KUKA KRL program: EPS_2_25452_SANMH01_A_20260112013754.src

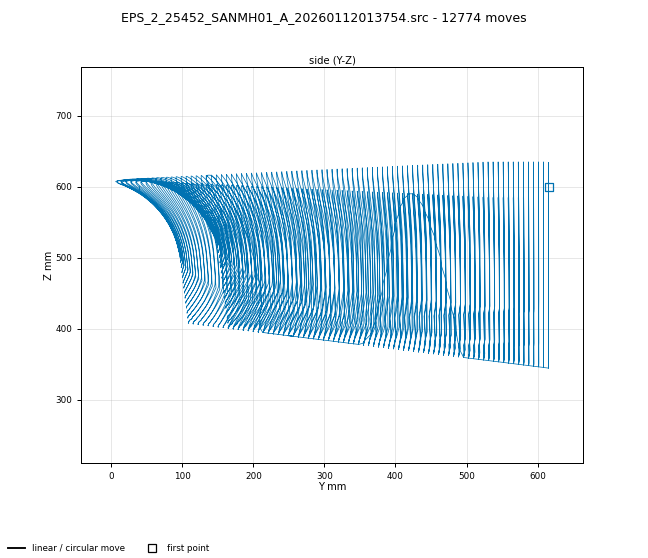
[picture p0: tool path of EPS_2_25452_SANMH01_A_20260112013754.src, 12774 of 12776 moves have a stored position in this frame; points joined in program order, loops and branches not executed]
&ACCESS RVP
&REL 4
&COMMENT QRS 19112012
&PARAM EDITMASK = *
DEF PART()
EXT BAS (BAS_COMMAND :IN,REAL :IN )
INT I
BAS (#INITMOV,0 )

;KUKA QRS Post kuka4.cps  Date:22-06-2017 !

File_ID=2960

QRS_PRE_INIT()

;Init var - Until changes are made in qrs_pre_init
Outlet_Square_prg=0
Inlet_1_Square_prg=0
Inlet_2_Square_prg=0
Inlet_3_Square_prg=0
Inlet_4_Square_prg=0
Inlet_5_Square_prg=0

Outlet_1={X 0.000, Y 530.070, Z 534.500, B 0.000, E1 0.000 }
Inlet_1={X 0.000, Y 533.640, Z 484.500, B 0.000, E1 171.000 }
Outlet_1_type=201
Inlet_1_type=201
;QRS#1=Sidecore dimensions
;QRS#2=200-8" PVC SDR 35
;QRS#3=200-8" PVC SDR 35
;QRS#4=
;QRS#5=
;QRS#6=
;QRS#7=
;QRS#8=
;QRS#9=12-08 PSX
;QRS#10=12-08 PSX
;QRS#11=
;QRS#12=
;QRS#13=
;QRS#14=
;QRS#15=
;QRS#16=1220x127x914 3'
;QRS#17=EPS Height
;QRS#18=635
;QRS#19=*
;QRS#20= UPDATED VERSION 22-06-2017
;QRS#21=*
Outlet_Square=0100
Inlet_1_Square=0100
Inlet_2_Square=0
Inlet_3_Square=0
Inlet_4_Square=0
Inlet_5_Square=0
Mill_Square=1
Outlet_Square_Prg=204
Inlet_1_Square_prg=204

QRS_INIT()

$ADVANCE=5

; T1
PTP {E1 173.589,E2 173.589}
PTP {X 0,Y 615.512,A -85,B 0,C 180,E1 173.589,E2 173.589,E3 0,E4 0,E5 0,E6 0}
QRS_SPEED_INIT()
LIN {X 0,Y 615.512,Z 600,A -85,B 0,C 180,E1 173.589,E2 173.589,E3 0,E4 0,E5 0,E6 0} C_VEL
LIN {X 0,Y 615.512,Z 354.868,A -85,B 0,C 180,E1 173.589,E2 173.589} C_VEL
LIN {X 0,Y 615.512,Z 346.696,A -85,B 0,C 180,E1 173.589,E2 173.589} C_VEL
LIN {X 0,Y 615.496,Z 344.696,A -85,B 0,C 180,E1 173.403,E2 173.403} C_VEL
LIN {X 0,Y 615.484,Z 344.688,A -85,B 0,C 180,E1 170.801,E2 170.801} C_VEL
LIN {X 0,Y 615.478,Z 344.686,A -85,B 0,C 180,E1 168.139,E2 168.139} C_VEL
LIN {X 0,Y 615.493,Z 344.701,A -85,B 0,C 180,E1 165.451,E2 165.451} C_VEL
LIN {X 0,Y 615.489,Z 344.683,A -85,B 0,C 180,E1 162.729,E2 162.729} C_VEL
LIN {X 0,Y 615.479,Z 344.691,A -85,B 0,C 180,E1 159.967,E2 159.967} C_VEL
LIN {X 0,Y 615.493,Z 344.699,A -85,B 0,C 180,E1 157.65,E2 157.65} C_VEL
LIN {X 0,Y 615.476,Z 344.688,A -85,B 0,C 180,E1 155.007,E2 155.007} C_VEL
LIN {X 0,Y 615.481,Z 344.684,A -85,B 0,C 180,E1 152.822,E2 152.822} C_VEL
LIN {X 0,Y 615.477,Z 344.691,A -85,B 0,C 180,E1 150.205,E2 150.205} C_VEL
LIN {X 0,Y 615.489,Z 344.694,A -85,B 0,C 180,E1 147.542,E2 147.542} C_VEL
LIN {X 0,Y 615.477,Z 344.687,A -85,B 0,C 180,E1 145.184,E2 145.184} C_VEL
LIN {X 0,Y 615.489,Z 344.683,A -85,B 0,C 180,E1 142.757,E2 142.757} C_VEL
LIN {X 0,Y 615.498,Z 344.699,A -85,B 0,C 180,E1 139.908,E2 139.908} C_VEL
LIN {X 0,Y 615.493,Z 344.69,A -85,B 0,C 180,E1 137.647,E2 137.647} C_VEL
LIN {X 0,Y 615.481,Z 344.684,A -85,B 0,C 180,E1 134.93,E2 134.93} C_VEL
LIN {X 0,Y 615.498,Z 344.7,A -85,B 0,C 180,E1 132.081,E2 132.081} C_VEL
LIN {X 0,Y 615.495,Z 344.688,A -85,B 0,C 180,E1 129.748,E2 129.748} C_VEL
LIN {X 0,Y 615.484,Z 344.685,A -85,B 0,C 180,E1 126.935,E2 126.935} C_VEL
LIN {X 0,Y 615.493,Z 344.693,A -85,B 0,C 180,E1 124.021,E2 124.021} C_VEL
LIN {X 0,Y 615.487,Z 344.685,A -85,B 0,C 180,E1 121.685,E2 121.685} C_VEL
LIN {X 0,Y 615.477,Z 344.685,A -85,B 0,C 180,E1 119.406,E2 119.406} C_VEL
LIN {X 0,Y 615.491,Z 344.805,A -85,B 0,C 180,E1 116.968,E2 116.968} C_VEL
LIN {X 0,Y 615.483,Z 360.204,A -85,B 0,C 180,E1 114.272,E2 114.272} C_VEL
LIN {X 0,Y 615.497,Z 374.44,A -85,B 0,C 180,E1 111.805,E2 111.805} C_VEL
LIN {X 0,Y 615.478,Z 480.331,A -85,B 0,C 180,E1 110.553,E2 110.553} C_VEL
LIN {X 0,Y 615.475,Z 493.827,A -85,B 0,C 180,E1 110.26,E2 110.26} C_VEL
LIN {X 0,Y 615.497,Z 506.182,A -85,B 0,C 180,E1 109.858,E2 109.858} C_VEL
LIN {X 0,Y 615.477,Z 518.044,A -85,B 0,C 180,E1 109.338,E2 109.338} C_VEL
LIN {X 0,Y 615.488,Z 528.758,A -85,B 0,C 180,E1 108.732,E2 108.732} C_VEL
LIN {X 0,Y 615.499,Z 539.692,A -85,B 0,C 180,E1 107.956,E2 107.956} C_VEL
LIN {X 0,Y 615.497,Z 549.463,A -85,B 0,C 180,E1 107.099,E2 107.099} C_VEL
LIN {X 0,Y 615.497,Z 557.985,A -85,B 0,C 180,E1 106.168,E2 106.168} C_VEL
LIN {X 0,Y 615.497,Z 565.024,A -85,B 0,C 180,E1 105.225,E2 105.225} C_VEL
LIN {X 0,Y 615.497,Z 570.956,A -85,B 0,C 180,E1 104.241,E2 104.241} C_VEL
LIN {X 0,Y 615.496,Z 575.897,A -85,B 0,C 180,E1 103.201,E2 103.201} C_VEL
LIN {X 0,Y 615.497,Z 579.504,A -85,B 0,C 180,E1 102.195,E2 102.195} C_VEL
LIN {X 0,Y 615.495,Z 582.657,A -85,B 0,C 180,E1 100.889,E2 100.889} C_VEL
LIN {X 0,Y 615.499,Z 583.995,A -85,B 0,C 180,E1 99.862,E2 99.862} C_VEL
LIN {X 0,Y 615.495,Z 584.296,A -85,B 0,C 180,E1 98.536,E2 98.536} C_VEL
LIN {X 0,Y 615.497,Z 583.85,A -85,B 0,C 180,E1 97.875,E2 97.875} C_VEL
LIN {X 0,Y 615.496,Z 581.72,A -85,B 0,C 180,E1 96.556,E2 96.556} C_VEL
LIN {X 0,Y 615.498,Z 579.037,A -85,B 0,C 180,E1 95.57,E2 95.57} C_VEL
LIN {X 0,Y 615.495,Z 575.36,A -85,B 0,C 180,E1 94.584,E2 94.584} C_VEL
LIN {X 0,Y 615.496,Z 570.584,A -85,B 0,C 180,E1 93.601,E2 93.601} C_VEL
LIN {X 0,Y 615.497,Z 564.573,A -85,B 0,C 180,E1 92.618,E2 92.618} C_VEL
LIN {X 0,Y 615.498,Z 557.116,A -85,B 0,C 180,E1 91.636,E2 91.636} C_VEL
LIN {X 0,Y 615.498,Z 549.527,A -85,B 0,C 180,E1 90.818,E2 90.818} C_VEL
LIN {X 0,Y 615.498,Z 539.238,A -85,B 0,C 180,E1 89.918,E2 89.918} C_VEL
LIN {X 0,Y 615.484,Z 528.822,A -85,B 0,C 180,E1 89.182,E2 89.182} C_VEL
LIN {X 0,Y 615.482,Z 517.116,A -85,B 0,C 180,E1 88.528,E2 88.528} C_VEL
LIN {X 0,Y 615.495,Z 504.679,A -85,B 0,C 180,E1 87.996,E2 87.996} C_VEL
LIN {X 0,Y 615.476,Z 493.022,A -85,B 0,C 180,E1 87.628,E2 87.628} C_VEL
LIN {X 0,Y 615.478,Z 480.616,A -85,B 0,C 180,E1 87.362,E2 87.362} C_VEL
LIN {X 0,Y 615.491,Z 374.366,A -85,B 0,C 180,E1 86.092,E2 86.092} C_VEL
LIN {X 0,Y 615.486,Z 358.994,A -85,B 0,C 180,E1 83.428,E2 83.428} C_VEL
LIN {X 0,Y 615.486,Z 344.686,A -85,B 0,C 180,E1 80.905,E2 80.905} C_VEL
LIN {X 0,Y 615.487,Z 344.686,A -85,B 0,C 180,E1 78.139,E2 78.139} C_VEL
LIN {X 0,Y 615.495,Z 344.696,A -85,B 0,C 180,E1 75.451,E2 75.451} C_VEL
LIN {X 0,Y 615.478,Z 344.685,A -85,B 0,C 180,E1 72.73,E2 72.73} C_VEL
LIN {X 0,Y 615.494,Z 344.692,A -85,B 0,C 180,E1 69.968,E2 69.968} C_VEL
LIN {X 0,Y 615.489,Z 344.685,A -85,B 0,C 180,E1 67.156,E2 67.156} C_VEL
LIN {X 0,Y 615.489,Z 344.688,A -85,B 0,C 180,E1 64.285,E2 64.285} C_VEL
LIN {X 0,Y 615.49,Z 344.687,A -85,B 0,C 180,E1 61.343,E2 61.343} C_VEL
LIN {X 0,Y 615.482,Z 344.684,A -85,B 0,C 180,E1 58.916,E2 58.916} C_VEL
LIN {X 0,Y 615.497,Z 344.7,A -85,B 0,C 180,E1 55.98,E2 55.98} C_VEL
LIN {X 0,Y 615.483,Z 344.684,A -85,B 0,C 180,E1 53.065,E2 53.065} C_VEL
LIN {X 0,Y 615.494,Z 344.695,A -85,B 0,C 180,E1 50.251,E2 50.251} C_VEL
LIN {X 0,Y 615.476,Z 344.691,A -85,B 0,C 180,E1 47.647,E2 47.647} C_VEL
LIN {X 0,Y 615.479,Z 344.685,A -85,B 0,C 180,E1 44.932,E2 44.932} C_VEL
LIN {X 0,Y 615.486,Z 344.698,A -85,B 0,C 180,E1 42.082,E2 42.082} C_VEL
LIN {X 0,Y 615.477,Z 344.69,A -85,B 0,C 180,E1 39.751,E2 39.751} C_VEL
LIN {X 0,Y 615.478,Z 344.687,A -85,B 0,C 180,E1 36.937,E2 36.937} C_VEL
LIN {X 0,Y 615.481,Z 344.693,A -85,B 0,C 180,E1 34.023,E2 34.023} C_VEL
LIN {X 0,Y 615.479,Z 344.686,A -85,B 0,C 180,E1 31.686,E2 31.686} C_VEL
LIN {X 0,Y 615.486,Z 344.683,A -85,B 0,C 180,E1 29.407,E2 29.407} C_VEL
LIN {X 0,Y 615.495,Z 344.699,A -85,B 0,C 180,E1 26.444,E2 26.444} C_VEL
LIN {X 0,Y 615.486,Z 344.683,A -85,B 0,C 180,E1 23.557,E2 23.557} C_VEL
LIN {X 0,Y 615.486,Z 344.698,A -85,B 0,C 180,E1 20.731,E2 20.731} C_VEL
LIN {X 0,Y 615.477,Z 344.687,A -85,B 0,C 180,E1 17.958,E2 17.958} C_VEL
LIN {X 0,Y 615.491,Z 344.686,A -85,B 0,C 180,E1 15.226,E2 15.226} C_VEL
LIN {X 0,Y 615.493,Z 344.694,A -85,B 0,C 180,E1 12.53,E2 12.53} C_VEL
LIN {X 0,Y 615.477,Z 344.685,A -85,B 0,C 180,E1 9.863,E2 9.863} C_VEL
LIN {X 0,Y 615.49,Z 344.69,A -85,B 0,C 180,E1 7.216,E2 7.216} C_VEL
LIN {X 0,Y 615.493,Z 344.691,A -85,B 0,C 180,E1 4.585,E2 4.585} C_VEL
LIN {X 0,Y 615.477,Z 344.685,A -85,B 0,C 180,E1 1.963,E2 1.963} C_VEL
LIN {X 0,Y 615.493,Z 344.69,A -85,B 0,C 180,E1 -0.654,E2 -0.654} C_VEL
LIN {X 0,Y 615.491,Z 344.691,A -85,B 0,C 180,E1 -3.273,E2 -3.273} C_VEL
LIN {X 0,Y 615.476,Z 344.685,A -85,B 0,C 180,E1 -5.899,E2 -5.899} C_VEL
LIN {X 0,Y 615.493,Z 344.691,A -85,B 0,C 180,E1 -8.536,E2 -8.536} C_VEL
LIN {X 0,Y 615.49,Z 344.69,A -85,B 0,C 180,E1 -11.193,E2 -11.193} C_VEL
LIN {X 0,Y 615.474,Z 344.686,A -85,B 0,C 180,E1 -13.933,E2 -13.933} C_VEL
LIN {X 0,Y 615.496,Z 344.696,A -85,B 0,C 180,E1 -16.586,E2 -16.586} C_VEL
LIN {X 0,Y 615.488,Z 344.685,A -85,B 0,C 180,E1 -19.338,E2 -19.338} C_VEL
LIN {X 0,Y 615.48,Z 344.69,A -85,B 0,C 180,E1 -22.137,E2 -22.137} C_VEL
LIN {X 0,Y 615.484,Z 344.69,A -85,B 0,C 180,E1 -24.992,E2 -24.992} C_VEL
LIN {X 0,Y 615.483,Z 344.686,A -85,B 0,C 180,E1 -27.177,E2 -27.177} C_VEL
LIN {X 0,Y 615.477,Z 344.687,A -85,B 0,C 180,E1 -29.795,E2 -29.795} C_VEL
LIN {X 0,Y 615.496,Z 344.7,A -85,B 0,C 180,E1 -32.457,E2 -32.457} C_VEL
LIN {X 0,Y 615.48,Z 344.691,A -85,B 0,C 180,E1 -34.816,E2 -34.816} C_VEL
LIN {X 0,Y 615.489,Z 344.682,A -85,B 0,C 180,E1 -37.242,E2 -37.242} C_VEL
LIN {X 0,Y 615.486,Z 344.696,A -85,B 0,C 180,E1 -40.09,E2 -40.09} C_VEL
LIN {X 0,Y 615.493,Z 344.697,A -85,B 0,C 180,E1 -42.353,E2 -42.353} C_VEL
LIN {X 0,Y 615.48,Z 344.684,A -85,B 0,C 180,E1 -45.069,E2 -45.069} C_VEL
LIN {X 0,Y 615.486,Z 344.696,A -85,B 0,C 180,E1 -47.92,E2 -47.92} C_VEL
LIN {X 0,Y 615.494,Z 344.695,A -85,B 0,C 180,E1 -50.252,E2 -50.252} C_VEL
LIN {X 0,Y 615.483,Z 344.684,A -85,B 0,C 180,E1 -53.064,E2 -53.064} C_VEL
LIN {X 0,Y 615.494,Z 344.701,A -85,B 0,C 180,E1 -55.979,E2 -55.979} C_VEL
LIN {X 0,Y 615.482,Z 344.684,A -85,B 0,C 180,E1 -58.915,E2 -58.915} C_VEL
LIN {X 0,Y 615.485,Z 344.692,A -85,B 0,C 180,E1 -61.551,E2 -61.551} C_VEL
LIN {X 0,Y 615.481,Z 344.687,A -85,B 0,C 180,E1 -64.433,E2 -64.433} C_VEL
LIN {X 0,Y 615.487,Z 344.827,A -85,B 0,C 180,E1 -67.067,E2 -67.067} C_VEL
LIN {X 0,Y 615.484,Z 366.758,A -85,B 0,C 180,E1 -69.968,E2 -69.968} C_VEL
LIN {X 0,Y 615.478,Z 388,A -85,B 0,C 180,E1 -72.73,E2 -72.73} C_VEL
LIN {X 0,Y 615.479,Z 409.218,A -85,B 0,C 180,E1 -75.451,E2 -75.451} C_VEL
LIN {X 0,Y 615.497,Z 422.298,A -85,B 0,C 180,E1 -77.114,E2 -77.114} C_VEL
LIN {X 0,Y 615.479,Z 530.847,A -85,B 0,C 180,E1 -78.411,E2 -78.411} C_VEL
LIN {X 0,Y 615.478,Z 543.355,A -85,B 0,C 180,E1 -78.682,E2 -78.682} C_VEL
LIN {X 0,Y 615.491,Z 556.568,A -85,B 0,C 180,E1 -79.111,E2 -79.111} C_VEL
LIN {X 0,Y 615.478,Z 568.483,A -85,B 0,C 180,E1 -79.639,E2 -79.639} C_VEL
LIN {X 0,Y 615.487,Z 579.999,A -85,B 0,C 180,E1 -80.304,E2 -80.304} C_VEL
LIN {X 0,Y 615.499,Z 590.344,A -85,B 0,C 180,E1 -81.05,E2 -81.05} C_VEL
LIN {X 0,Y 615.497,Z 598.814,A -85,B 0,C 180,E1 -81.794,E2 -81.794} C_VEL
LIN {X 0,Y 615.498,Z 606.608,A -85,B 0,C 180,E1 -82.62,E2 -82.62} C_VEL
LIN {X 0,Y 615.496,Z 614.204,A -85,B 0,C 180,E1 -83.608,E2 -83.608} C_VEL
LIN {X 0,Y 615.498,Z 621.205,A -85,B 0,C 180,E1 -84.759,E2 -84.759} C_VEL
LIN {X 0,Y 615.493,Z 625.852,A -85,B 0,C 180,E1 -85.744,E2 -85.744} C_VEL
LIN {X 0,Y 615.495,Z 629.399,A -85,B 0,C 180,E1 -86.727,E2 -86.727} C_VEL
LIN {X 0,Y 615.497,Z 631.233,A -85,B 0,C 180,E1 -87.382,E2 -87.382} C_VEL
LIN {X 0,Y 615.497,Z 632.608,A -85,B 0,C 180,E1 -88.037,E2 -88.037} C_VEL
LIN {X 0,Y 615.496,Z 634.174,A -85,B 0,C 180,E1 -89.346,E2 -89.346} C_VEL
LIN {X 0,Y 615.494,Z 634.389,A -85,B 0,C 180,E1 -90,E2 -90} C_VEL
LIN {X 0,Y 615.496,Z 633.58,A -85,B 0,C 180,E1 -91.309,E2 -91.309} C_VEL
LIN {X 0,Y 615.497,Z 632.608,A -85,B 0,C 180,E1 -91.963,E2 -91.963} C_VEL
LIN {X 0,Y 615.497,Z 631.233,A -85,B 0,C 180,E1 -92.618,E2 -92.618} C_VEL
LIN {X 0,Y 615.496,Z 628.35,A -85,B 0,C 180,E1 -93.601,E2 -93.601} C_VEL
LIN {X 0,Y 615.498,Z 624.442,A -85,B 0,C 180,E1 -94.584,E2 -94.584} C_VEL
LIN {X 0,Y 615.499,Z 619.406,A -85,B 0,C 180,E1 -95.57,E2 -95.57} C_VEL
LIN {X 0,Y 615.497,Z 612.869,A -85,B 0,C 180,E1 -96.583,E2 -96.583} C_VEL
LIN {X 0,Y 615.497,Z 605.135,A -85,B 0,C 180,E1 -97.545,E2 -97.545} C_VEL
LIN {X 0,Y 615.498,Z 597.047,A -85,B 0,C 180,E1 -98.371,E2 -98.371} C_VEL
LIN {X 0,Y 615.499,Z 587.17,A -85,B 0,C 180,E1 -99.198,E2 -99.198} C_VEL
LIN {X 0,Y 615.488,Z 575.985,A -85,B 0,C 180,E1 -99.945,E2 -99.945} C_VEL
LIN {X 0,Y 615.481,Z 565.029,A -85,B 0,C 180,E1 -100.527,E2 -100.527} C_VEL
LIN {X 0,Y 615.49,Z 552.452,A -85,B 0,C 180,E1 -101.041,E2 -101.041} C_VEL
LIN {X 0,Y 615.477,Z 540.079,A -85,B 0,C 180,E1 -101.401,E2 -101.401} C_VEL
LIN {X 0,Y 615.481,Z 526.487,A -85,B 0,C 180,E1 -101.652,E2 -101.652} C_VEL
LIN {X 0,Y 615.497,Z 422.298,A -85,B 0,C 180,E1 -102.886,E2 -102.886} C_VEL
LIN {X 0,Y 615.485,Z 399.937,A -85,B 0,C 180,E1 -105.735,E2 -105.735} C_VEL
LIN {X 0,Y 615.481,Z 377.716,A -85,B 0,C 180,E1 -108.602,E2 -108.602} C_VEL
LIN {X 0,Y 615.478,Z 357.457,A -85,B 0,C 180,E1 -111.256,E2 -111.256} C_VEL
LIN {X 0,Y 615.486,Z 344.684,A -85,B 0,C 180,E1 -112.977,E2 -112.977} C_VEL
LIN {X 0,Y 615.489,Z 344.689,A -85,B 0,C 180,E1 -115.715,E2 -115.715} C_VEL
LIN {X 0,Y 615.488,Z 344.686,A -85,B 0,C 180,E1 -118.657,E2 -118.657} C_VEL
LIN {X 0,Y 615.482,Z 344.684,A -85,B 0,C 180,E1 -121.085,E2 -121.085} C_VEL
LIN {X 0,Y 615.494,Z 344.7,A -85,B 0,C 180,E1 -124.021,E2 -124.021} C_VEL
LIN {X 0,Y 615.483,Z 344.684,A -85,B 0,C 180,E1 -126.936,E2 -126.936} C_VEL
LIN {X 0,Y 615.494,Z 344.697,A -85,B 0,C 180,E1 -129.748,E2 -129.748} C_VEL
LIN {X 0,Y 615.478,Z 344.689,A -85,B 0,C 180,E1 -132.353,E2 -132.353} C_VEL
LIN {X 0,Y 615.48,Z 344.686,A -85,B 0,C 180,E1 -135.068,E2 -135.068} C_VEL
LIN {X 0,Y 615.486,Z 344.696,A -85,B 0,C 180,E1 -137.918,E2 -137.918} C_VEL
LIN {X 0,Y 615.477,Z 344.689,A -85,B 0,C 180,E1 -140.249,E2 -140.249} C_VEL
LIN {X 0,Y 615.482,Z 344.688,A -85,B 0,C 180,E1 -143.062,E2 -143.062} C_VEL
LIN {X 0,Y 615.481,Z 344.691,A -85,B 0,C 180,E1 -145.978,E2 -145.978} C_VEL
LIN {X 0,Y 615.479,Z 344.685,A -85,B 0,C 180,E1 -148.314,E2 -148.314} C_VEL
LIN {X 0,Y 615.487,Z 344.683,A -85,B 0,C 180,E1 -150.594,E2 -150.594} C_VEL
LIN {X 0,Y 615.497,Z 344.695,A -85,B 0,C 180,E1 -153.556,E2 -153.556} C_VEL
LIN {X 0,Y 615.486,Z 344.683,A -85,B 0,C 180,E1 -156.444,E2 -156.444} C_VEL
LIN {X 0,Y 615.495,Z 344.701,A -85,B 0,C 180,E1 -159.27,E2 -159.27} C_VEL
LIN {X 0,Y 615.477,Z 344.686,A -85,B 0,C 180,E1 -162.043,E2 -162.043} C_VEL
LIN {X 0,Y 615.492,Z 344.689,A -85,B 0,C 180,E1 -164.774,E2 -164.774} C_VEL
LIN {X 0,Y 615.491,Z 344.69,A -85,B 0,C 180,E1 -167.47,E2 -167.47} C_VEL
LIN {X 0,Y 615.477,Z 344.685,A -85,B 0,C 180,E1 -170.138,E2 -170.138} C_VEL
LIN {X 0,Y 615.495,Z 344.693,A -85,B 0,C 180,E1 -172.785,E2 -172.785} C_VEL
LIN {X 0,Y 615.491,Z 344.688,A -85,B 0,C 180,E1 -175.416,E2 -175.416} C_VEL
LIN {X 0,Y 615.477,Z 344.685,A -85,B 0,C 180,E1 -178.037,E2 -178.037} C_VEL
LIN {X 0,Y 615.495,Z 344.694,A -85,B 0,C 180,E1 -180.654,E2 -180.654} C_VEL
LIN {X 0,Y 615.491,Z 344.687,A -85,B 0,C 180,E1 -183.273,E2 -183.273} C_VEL
LIN {X 0,Y 615.476,Z 344.686,A -85,B 0,C 180,E1 -185.899,E2 -185.899} C_VEL
LIN {X 0,Y 615.496,Z 344.696,A -85,B 0,C 180,E1 -186.597,E2 -186.597} C_VEL
LIN {X 0,Y 614.815,Z 344.835,A -85,B 0,C 180,E1 -187.143,E2 -187.143} C_VEL
LIN {X 0,Y 611.975,Z 345.25,A -85,B 0,C 180,E1 -188.028,E2 -188.028} C_VEL
LIN {X 0,Y 609.58,Z 345.56,A -85,B 0,C 180,E1 -188.741,E2 -188.741} C_VEL
LIN {X 0,Y 608.544,Z 345.678,A -85,B 0,C 180,E1 -189.291,E2 -189.291} C_VEL
LIN {X 0,Y 608.454,Z 345.688,A -85,B 0,C 180,E1 -189.477,E2 -189.477} C_VEL
LIN {X 0,Y 608.456,Z 345.689,A -85,B 0,C 180,E1 -192,E2 -192} C_VEL
LIN {X 0,Y 608.478,Z 345.692,A -85,B 0,C 180,E1 -194.721,E2 -194.721} C_VEL
LIN {X 0,Y 608.451,Z 345.688,A -85,B 0,C 180,E1 -197.477,E2 -197.477} C_VEL
LIN {X 0,Y 608.46,Z 345.694,A -85,B 0,C 180,E1 -200.275,E2 -200.275} C_VEL
LIN {X 0,Y 608.456,Z 345.697,A -85,B 0,C 180,E1 -202.479,E2 -202.479} C_VEL
LIN {X 0,Y 608.45,Z 345.695,A -85,B 0,C 180,E1 -204.572,E2 -204.572} C_VEL
LIN {X 0,Y 608.473,Z 345.685,A -85,B 0,C 180,E1 -207.209,E2 -207.209} C_VEL
LIN {X 0,Y 608.461,Z 345.692,A -85,B 0,C 180,E1 -209.973,E2 -209.973} C_VEL
LIN {X 0,Y 608.462,Z 345.691,A -85,B 0,C 180,E1 -212.525,E2 -212.525} C_VEL
LIN {X 0,Y 608.439,Z 345.689,A -85,B 0,C 180,E1 -215.278,E2 -215.278} C_VEL
LIN {X 0,Y 608.473,Z 345.69,A -85,B 0,C 180,E1 -217.747,E2 -217.747} C_VEL
LIN {X 0,Y 608.478,Z 345.69,A -85,B 0,C 180,E1 -220.334,E2 -220.334} C_VEL
LIN {X 0,Y 608.484,Z 345.685,A -85,B 0,C 180,E1 -223.312,E2 -223.312} C_VEL
LIN {X 0,Y 608.477,Z 345.692,A -85,B 0,C 180,E1 -226.133,E2 -226.133} C_VEL
LIN {X 0,Y 608.45,Z 345.688,A -85,B 0,C 180,E1 -228.824,E2 -228.824} C_VEL
LIN {X 0,Y 608.473,Z 345.689,A -85,B 0,C 180,E1 -231.413,E2 -231.413} C_VEL
LIN {X 0,Y 608.48,Z 345.692,A -85,B 0,C 180,E1 -233.951,E2 -233.951} C_VEL
LIN {X 0,Y 608.463,Z 345.688,A -85,B 0,C 180,E1 -236.33,E2 -236.33} C_VEL
LIN {X 0,Y 608.448,Z 345.688,A -85,B 0,C 180,E1 -238.733,E2 -238.733} C_VEL
LIN {X 0,Y 608.482,Z 345.69,A -85,B 0,C 180,E1 -241.38,E2 -241.38} C_VEL
LIN {X 0,Y 608.479,Z 345.704,A -85,B 0,C 180,E1 -242.962,E2 -242.962} C_VEL
LIN {X 0,Y 608.478,Z 362.057,A -85,B 0,C 180,E1 -245.849,E2 -245.849} C_VEL
LIN {X 0,Y 608.467,Z 374.632,A -85,B 0,C 180,E1 -248.042,E2 -248.042} C_VEL
LIN {X 0,Y 608.53,Z 481.606,A -85,B 0,C 180,E1 -249.333,E2 -249.333} C_VEL
LIN {X 0,Y 608.52,Z 495.277,A -85,B 0,C 180,E1 -249.646,E2 -249.646} C_VEL
LIN {X 0,Y 608.52,Z 508.023,A -85,B 0,C 180,E1 -250.081,E2 -250.081} C_VEL
LIN {X 0,Y 608.505,Z 519.44,A -85,B 0,C 180,E1 -250.607,E2 -250.607} C_VEL
LIN {X 0,Y 608.471,Z 530.955,A -85,B 0,C 180,E1 -251.286,E2 -251.286} C_VEL
LIN {X 0,Y 608.478,Z 541.839,A -85,B 0,C 180,E1 -252.09,E2 -252.09} C_VEL
LIN {X 0,Y 608.462,Z 552.081,A -85,B 0,C 180,E1 -253.044,E2 -253.044} C_VEL
LIN {X 0,Y 608.462,Z 560.996,A -85,B 0,C 180,E1 -254.079,E2 -254.079} C_VEL
LIN {X 0,Y 608.451,Z 568.049,A -85,B 0,C 180,E1 -255.108,E2 -255.108} C_VEL
LIN {X 0,Y 608.432,Z 574.549,A -85,B 0,C 180,E1 -256.319,E2 -256.319} C_VEL
LIN {X 0,Y 608.428,Z 578.613,A -85,B 0,C 180,E1 -257.322,E2 -257.322} C_VEL
LIN {X 0,Y 608.445,Z 580.752,A -85,B 0,C 180,E1 -258,E2 -258} C_VEL
LIN {X 0,Y 608.423,Z 583.219,A -85,B 0,C 180,E1 -259.07,E2 -259.07} C_VEL
LIN {X 0,Y 608.434,Z 584.527,A -85,B 0,C 180,E1 -260.023,E2 -260.023} C_VEL
LIN {X 0,Y 608.419,Z 584.931,A -85,B 0,C 180,E1 -261.364,E2 -261.364} C_VEL
LIN {X 0,Y 608.422,Z 584.554,A -85,B 0,C 180,E1 -262.033,E2 -262.033} C_VEL
LIN {X 0,Y 608.421,Z 583.75,A -85,B 0,C 180,E1 -262.7,E2 -262.7} C_VEL
LIN {X 0,Y 608.449,Z 582.463,A -85,B 0,C 180,E1 -263.398,E2 -263.398} C_VEL
LIN {X 0,Y 608.442,Z 578.86,A -85,B 0,C 180,E1 -264.698,E2 -264.698} C_VEL
LIN {X 0,Y 608.441,Z 574.9,A -85,B 0,C 180,E1 -265.694,E2 -265.694} C_VEL
LIN {X 0,Y 608.458,Z 568.82,A -85,B 0,C 180,E1 -266.855,E2 -266.855} C_VEL
LIN {X 0,Y 608.454,Z 562.203,A -85,B 0,C 180,E1 -267.849,E2 -267.849} C_VEL
LIN {X 0,Y 608.479,Z 554.016,A -85,B 0,C 180,E1 -268.842,E2 -268.842} C_VEL
LIN {X 0,Y 608.469,Z 545.669,A -85,B 0,C 180,E1 -269.669,E2 -269.669} C_VEL
LIN {X 0,Y 608.479,Z 535.396,A -85,B 0,C 180,E1 -270.496,E2 -270.496} C_VEL
LIN {X 0,Y 608.485,Z 523.897,A -85,B 0,C 180,E1 -271.241,E2 -271.241} C_VEL
LIN {X 0,Y 608.502,Z 512.472,A -85,B 0,C 180,E1 -271.82,E2 -271.82} C_VEL
LIN {X 0,Y 608.512,Z 499.459,A -85,B 0,C 180,E1 -272.317,E2 -272.317} C_VEL
LIN {X 0,Y 608.521,Z 486.295,A -85,B 0,C 180,E1 -272.668,E2 -272.668} C_VEL
LIN {X 0,Y 608.536,Z 471.453,A -85,B 0,C 180,E1 -272.896,E2 -272.896} C_VEL
LIN {X 0,Y 608.537,Z 375.202,A -85,B 0,C 180,E1 -274.036,E2 -274.036} C_VEL
LIN {X 0,Y 608.458,Z 374.585,A -85,B 0,C 180,E1 -274.057,E2 -274.057} C_VEL
LIN {X 0,Y 608.486,Z 357.93,A -85,B 0,C 180,E1 -276.966,E2 -276.966} C_VEL
LIN {X 0,Y 608.477,Z 345.686,A -85,B 0,C 180,E1 -279.138,E2 -279.138} C_VEL
LIN {X 0,Y 608.465,Z 345.689,A -85,B 0,C 180,E1 -281.999,E2 -281.999} C_VEL
LIN {X 0,Y 608.48,Z 345.689,A -85,B 0,C 180,E1 -284.72,E2 -284.72} C_VEL
LIN {X 0,Y 608.452,Z 345.688,A -85,B 0,C 180,E1 -287.476,E2 -287.476} C_VEL
LIN {X 0,Y 608.47,Z 345.696,A -85,B 0,C 180,E1 -290.273,E2 -290.273} C_VEL
LIN {X 0,Y 608.451,Z 345.688,A -85,B 0,C 180,E1 -293.123,E2 -293.123} C_VEL
LIN {X 0,Y 608.472,Z 345.688,A -85,B 0,C 180,E1 -295.72,E2 -295.72} C_VEL
LIN {X 0,Y 608.476,Z 345.687,A -85,B 0,C 180,E1 -298.619,E2 -298.619} C_VEL
LIN {X 0,Y 608.447,Z 345.689,A -85,B 0,C 180,E1 -301.317,E2 -301.317} C_VEL
LIN {X 0,Y 608.473,Z 345.69,A -85,B 0,C 180,E1 -303.734,E2 -303.734} C_VEL
LIN {X 0,Y 608.479,Z 345.694,A -85,B 0,C 180,E1 -306.089,E2 -306.089} C_VEL
LIN {X 0,Y 608.471,Z 345.687,A -85,B 0,C 180,E1 -308.587,E2 -308.587} C_VEL
LIN {X 0,Y 608.457,Z 345.689,A -85,B 0,C 180,E1 -311.341,E2 -311.341} C_VEL
LIN {X 0,Y 608.449,Z 345.692,A -85,B 0,C 180,E1 -314.263,E2 -314.263} C_VEL
LIN {X 0,Y 608.453,Z 345.688,A -85,B 0,C 180,E1 -317.04,E2 -317.04} C_VEL
LIN {X 0,Y 608.449,Z 345.698,A -85,B 0,C 180,E1 -319.696,E2 -319.696} C_VEL
LIN {X 0,Y 608.467,Z 345.688,A -85,B 0,C 180,E1 -322.253,E2 -322.253} C_VEL
LIN {X 0,Y 608.436,Z 345.69,A -85,B 0,C 180,E1 -324.721,E2 -324.721} C_VEL
LIN {X 0,Y 608.466,Z 345.694,A -85,B 0,C 180,E1 -327.475,E2 -327.475} C_VEL
LIN {X 0,Y 608.462,Z 345.688,A -85,B 0,C 180,E1 -330.22,E2 -330.22} C_VEL
LIN {X 0,Y 608.475,Z 345.685,A -85,B 0,C 180,E1 -332.791,E2 -332.791} C_VEL
LIN {X 0,Y 608.453,Z 345.698,A -85,B 0,C 180,E1 -335.429,E2 -335.429} C_VEL
LIN {X 0,Y 608.47,Z 345.685,A -85,B 0,C 180,E1 -338.308,E2 -338.308} C_VEL
LIN {X 0,Y 608.472,Z 345.695,A -85,B 0,C 180,E1 -341.28,E2 -341.28} C_VEL
LIN {X 0,Y 608.457,Z 345.689,A -85,B 0,C 180,E1 -343.906,E2 -343.906} C_VEL
LIN {X 0,Y 608.464,Z 345.688,A -85,B 0,C 180,E1 -346.643,E2 -346.643} C_VEL
LIN {X 0,Y 608.474,Z 345.693,A -85,B 0,C 180,E1 -349.35,E2 -349.35} C_VEL
LIN {X 0,Y 608.471,Z 345.685,A -85,B 0,C 180,E1 -352.033,E2 -352.033} C_VEL
LIN {X 0,Y 608.469,Z 345.689,A -85,B 0,C 180,E1 -354.698,E2 -354.698} C_VEL
LIN {X 0,Y 608.485,Z 345.689,A -85,B 0,C 180,E1 -357.352,E2 -357.352} C_VEL
LIN {X 0,Y 608.468,Z 345.686,A -85,B 0,C 180,E1 -360,E2 -360} C_VEL
LIN {X 0,Y 608.485,Z 345.689,A -85,B 0,C 180,E1 -362.648,E2 -362.648} C_VEL
LIN {X 0,Y 608.47,Z 345.689,A -85,B 0,C 180,E1 -365.302,E2 -365.302} C_VEL
LIN {X 0,Y 608.471,Z 345.685,A -85,B 0,C 180,E1 -367.967,E2 -367.967} C_VEL
LIN {X 0,Y 608.473,Z 345.693,A -85,B 0,C 180,E1 -370.65,E2 -370.65} C_VEL
LIN {X 0,Y 608.464,Z 345.688,A -85,B 0,C 180,E1 -373.356,E2 -373.356} C_VEL
LIN {X 0,Y 608.457,Z 345.688,A -85,B 0,C 180,E1 -376.094,E2 -376.094} C_VEL
LIN {X 0,Y 608.456,Z 345.694,A -85,B 0,C 180,E1 -378.87,E2 -378.87} C_VEL
LIN {X 0,Y 608.47,Z 345.685,A -85,B 0,C 180,E1 -381.691,E2 -381.691} C_VEL
LIN {X 0,Y 608.453,Z 345.698,A -85,B 0,C 180,E1 -384.571,E2 -384.571} C_VEL
LIN {X 0,Y 608.475,Z 345.686,A -85,B 0,C 180,E1 -387.209,E2 -387.209} C_VEL
LIN {X 0,Y 608.46,Z 345.689,A -85,B 0,C 180,E1 -389.973,E2 -389.973} C_VEL
LIN {X 0,Y 608.468,Z 345.694,A -85,B 0,C 180,E1 -392.525,E2 -392.525} C_VEL
LIN {X 0,Y 608.438,Z 345.689,A -85,B 0,C 180,E1 -395.278,E2 -395.278} C_VEL
LIN {X 0,Y 608.467,Z 345.688,A -85,B 0,C 180,E1 -397.746,E2 -397.746} C_VEL
LIN {X 0,Y 608.449,Z 345.698,A -85,B 0,C 180,E1 -400.33,E2 -400.33} C_VEL
LIN {X 0,Y 608.483,Z 345.684,A -85,B 0,C 180,E1 -403.312,E2 -403.312} C_VEL
LIN {X 0,Y 608.467,Z 345.696,A -85,B 0,C 180,E1 -406.132,E2 -406.132} C_VEL
LIN {X 0,Y 608.45,Z 345.689,A -85,B 0,C 180,E1 -408.824,E2 -408.824} C_VEL
LIN {X 0,Y 608.47,Z 345.687,A -85,B 0,C 180,E1 -411.413,E2 -411.413} C_VEL
LIN {X 0,Y 608.478,Z 345.694,A -85,B 0,C 180,E1 -413.951,E2 -413.951} C_VEL
LIN {X 0,Y 608.463,Z 345.691,A -85,B 0,C 180,E1 -416.33,E2 -416.33} C_VEL
LIN {X 0,Y 608.476,Z 345.685,A -85,B 0,C 180,E1 -418.728,E2 -418.728} C_VEL
LIN {X 0,Y 608.474,Z 345.687,A -85,B 0,C 180,E1 -421.38,E2 -421.38} C_VEL
LIN {X 0,Y 608.471,Z 345.689,A -85,B 0,C 180,E1 -424.28,E2 -424.28} C_VEL
LIN {X 0,Y 608.479,Z 345.824,A -85,B 0,C 180,E1 -426.923,E2 -426.923} C_VEL
LIN {X 0,Y 608.582,Z 361.447,A -85,B 0,C 180,E1 -429.024,E2 -429.024} C_VEL
LIN {X 0,Y 608.518,Z 382.72,A -85,B 0,C 180,E1 -431.831,E2 -431.831} C_VEL
LIN {X 0,Y 608.492,Z 402.663,A -85,B 0,C 180,E1 -434.423,E2 -434.423} C_VEL
LIN {X 0,Y 608.503,Z 422.524,A -85,B 0,C 180,E1 -436.974,E2 -436.974} C_VEL
LIN {X 0,Y 608.538,Z 530.962,A -85,B 0,C 180,E1 -438.277,E2 -438.277} C_VEL
LIN {X 0,Y 608.514,Z 544.226,A -85,B 0,C 180,E1 -438.572,E2 -438.572} C_VEL
LIN {X 0,Y 608.517,Z 556.598,A -85,B 0,C 180,E1 -438.981,E2 -438.981} C_VEL
LIN {X 0,Y 608.498,Z 568.639,A -85,B 0,C 180,E1 -439.519,E2 -439.519} C_VEL
LIN {X 0,Y 608.48,Z 580.201,A -85,B 0,C 180,E1 -440.191,E2 -440.191} C_VEL
LIN {X 0,Y 608.485,Z 590.596,A -85,B 0,C 180,E1 -440.946,E2 -440.946} C_VEL
LIN {X 0,Y 608.475,Z 599.114,A -85,B 0,C 180,E1 -441.699,E2 -441.699} C_VEL
LIN {X 0,Y 608.471,Z 606.962,A -85,B 0,C 180,E1 -442.534,E2 -442.534} C_VEL
LIN {X 0,Y 608.46,Z 614.287,A -85,B 0,C 180,E1 -443.485,E2 -443.485} C_VEL
LIN {X 0,Y 608.45,Z 619.867,A -85,B 0,C 180,E1 -444.366,E2 -444.366} C_VEL
LIN {X 0,Y 608.432,Z 624.951,A -85,B 0,C 180,E1 -445.362,E2 -445.362} C_VEL
LIN {X 0,Y 608.449,Z 628.896,A -85,B 0,C 180,E1 -446.358,E2 -446.358} C_VEL
LIN {X 0,Y 608.425,Z 631.809,A -85,B 0,C 180,E1 -447.352,E2 -447.352} C_VEL
LIN {X 0,Y 608.442,Z 633.201,A -85,B 0,C 180,E1 -448.014,E2 -448.014} C_VEL
LIN {X 0,Y 608.438,Z 634.783,A -85,B 0,C 180,E1 -449.338,E2 -449.338} C_VEL
LIN {X 0,Y 608.434,Z 635,A -85,B 0,C 180,E1 -450,E2 -450} C_VEL
LIN {X 0,Y 608.448,Z 634.184,A -85,B 0,C 180,E1 -451.324,E2 -451.324} C_VEL
LIN {X 0,Y 608.442,Z 633.201,A -85,B 0,C 180,E1 -451.986,E2 -451.986} C_VEL
LIN {X 0,Y 608.425,Z 631.809,A -85,B 0,C 180,E1 -452.648,E2 -452.648} C_VEL
LIN {X 0,Y 608.449,Z 628.896,A -85,B 0,C 180,E1 -453.642,E2 -453.642} C_VEL
LIN {X 0,Y 608.432,Z 624.95,A -85,B 0,C 180,E1 -454.638,E2 -454.638} C_VEL
LIN {X 0,Y 608.437,Z 618.877,A -85,B 0,C 180,E1 -455.801,E2 -455.801} C_VEL
LIN {X 0,Y 608.462,Z 612.236,A -85,B 0,C 180,E1 -456.799,E2 -456.799} C_VEL
LIN {X 0,Y 608.455,Z 603.991,A -85,B 0,C 180,E1 -457.8,E2 -457.8} C_VEL
LIN {X 0,Y 608.472,Z 595.538,A -85,B 0,C 180,E1 -458.636,E2 -458.636} C_VEL
LIN {X 0,Y 608.471,Z 585.094,A -85,B 0,C 180,E1 -459.473,E2 -459.473} C_VEL
LIN {X 0,Y 608.494,Z 574.76,A -85,B 0,C 180,E1 -460.144,E2 -460.144} C_VEL
LIN {X 0,Y 608.521,Z 563.255,A -85,B 0,C 180,E1 -460.74,E2 -460.74} C_VEL
LIN {X 0,Y 608.531,Z 550.887,A -85,B 0,C 180,E1 -461.225,E2 -461.225} C_VEL
LIN {X 0,Y 608.537,Z 537.45,A -85,B 0,C 180,E1 -461.597,E2 -461.597} C_VEL
LIN {X 0,Y 608.546,Z 525.105,A -85,B 0,C 180,E1 -461.808,E2 -461.808} C_VEL
LIN {X 0,Y 608.493,Z 422.441,A -85,B 0,C 180,E1 -463.037,E2 -463.037} C_VEL
LIN {X 0,Y 608.494,Z 400.004,A -85,B 0,C 180,E1 -465.92,E2 -465.92} C_VEL
LIN {X 0,Y 608.54,Z 378.405,A -85,B 0,C 180,E1 -468.735,E2 -468.735} C_VEL
LIN {X 0,Y 608.563,Z 357.458,A -85,B 0,C 180,E1 -471.51,E2 -471.51} C_VEL
LIN {X 0,Y 608.468,Z 345.688,A -85,B 0,C 180,E1 -473.1,E2 -473.1} C_VEL
LIN {X 0,Y 608.471,Z 345.689,A -85,B 0,C 180,E1 -475.72,E2 -475.72} C_VEL
LIN {X 0,Y 608.474,Z 345.687,A -85,B 0,C 180,E1 -478.62,E2 -478.62} C_VEL
LIN {X 0,Y 608.475,Z 345.685,A -85,B 0,C 180,E1 -481.315,E2 -481.315} C_VEL
LIN {X 0,Y 608.472,Z 345.691,A -85,B 0,C 180,E1 -483.734,E2 -483.734} C_VEL
LIN {X 0,Y 608.476,Z 345.693,A -85,B 0,C 180,E1 -486.089,E2 -486.089} C_VEL
LIN {X 0,Y 608.47,Z 345.686,A -85,B 0,C 180,E1 -488.587,E2 -488.587} C_VEL
LIN {X 0,Y 608.457,Z 345.69,A -85,B 0,C 180,E1 -491.341,E2 -491.341} C_VEL
LIN {X 0,Y 608.449,Z 345.691,A -85,B 0,C 180,E1 -494.263,E2 -494.263} C_VEL
LIN {X 0,Y 608.453,Z 345.688,A -85,B 0,C 180,E1 -497.04,E2 -497.04} C_VEL
LIN {X 0,Y 608.45,Z 345.698,A -85,B 0,C 180,E1 -499.696,E2 -499.696} C_VEL
LIN {X 0,Y 608.467,Z 345.687,A -85,B 0,C 180,E1 -502.254,E2 -502.254} C_VEL
LIN {X 0,Y 608.473,Z 345.688,A -85,B 0,C 180,E1 -505.089,E2 -505.089} C_VEL
LIN {X 0,Y 608.47,Z 345.689,A -85,B 0,C 180,E1 -507.906,E2 -507.906} C_VEL
LIN {X 0,Y 608.462,Z 345.687,A -85,B 0,C 180,E1 -510.22,E2 -510.22} C_VEL
LIN {X 0,Y 608.476,Z 345.686,A -85,B 0,C 180,E1 -512.791,E2 -512.791} C_VEL
LIN {X 0,Y 608.454,Z 345.697,A -85,B 0,C 180,E1 -515.429,E2 -515.429} C_VEL
LIN {X 0,Y 608.47,Z 345.685,A -85,B 0,C 180,E1 -518.309,E2 -518.309} C_VEL
LIN {X 0,Y 608.472,Z 345.695,A -85,B 0,C 180,E1 -521.28,E2 -521.28} C_VEL
LIN {X 0,Y 608.457,Z 345.688,A -85,B 0,C 180,E1 -523.906,E2 -523.906} C_VEL
LIN {X 0,Y 608.465,Z 345.689,A -85,B 0,C 180,E1 -526.644,E2 -526.644} C_VEL
LIN {X 0,Y 608.472,Z 345.691,A -85,B 0,C 180,E1 -529.35,E2 -529.35} C_VEL
LIN {X 0,Y 608.47,Z 345.685,A -85,B 0,C 180,E1 -532.033,E2 -532.033} C_VEL
LIN {X 0,Y 608.471,Z 345.691,A -85,B 0,C 180,E1 -534.698,E2 -534.698} C_VEL
LIN {X 0,Y 608.483,Z 345.687,A -85,B 0,C 180,E1 -537.352,E2 -537.352} C_VEL
LIN {X 0,Y 608.468,Z 345.686,A -85,B 0,C 180,E1 -540,E2 -540} C_VEL
LIN {X 0,Y 608.486,Z 345.691,A -85,B 0,C 180,E1 -542.648,E2 -542.648} C_VEL
LIN {X 0,Y 608.467,Z 345.688,A -85,B 0,C 180,E1 -545.302,E2 -545.302} C_VEL
LIN {X 0,Y 608.471,Z 345.686,A -85,B 0,C 180,E1 -547.967,E2 -547.967} C_VEL
LIN {X 0,Y 608.454,Z 345.688,A -85,B 0,C 180,E1 -549.477,E2 -549.477} C_VEL
LIN {X 0,Y 607.774,Z 345.774,A -85,B 0,C 180,E1 -550.029,E2 -550.029} C_VEL
LIN {X 0,Y 604.917,Z 346.133,A -85,B 0,C 180,E1 -550.926,E2 -550.926} C_VEL
LIN {X 0,Y 602.516,Z 346.431,A -85,B 0,C 180,E1 -551.648,E2 -551.648} C_VEL
LIN {X 0,Y 601.49,Z 346.559,A -85,B 0,C 180,E1 -552.205,E2 -552.205} C_VEL
LIN {X 0,Y 601.408,Z 346.568,A -85,B 0,C 180,E1 -552.393,E2 -552.393} C_VEL
LIN {X 0,Y 601.43,Z 346.567,A -85,B 0,C 180,E1 -554.897,E2 -554.897} C_VEL
LIN {X 0,Y 601.428,Z 346.566,A -85,B 0,C 180,E1 -556.986,E2 -556.986} C_VEL
LIN {X 0,Y 601.403,Z 346.567,A -85,B 0,C 180,E1 -559.81,E2 -559.81} C_VEL
LIN {X 0,Y 601.409,Z 346.572,A -85,B 0,C 180,E1 -562.607,E2 -562.607} C_VEL
LIN {X 0,Y 601.398,Z 346.568,A -85,B 0,C 180,E1 -564.879,E2 -564.879} C_VEL
LIN {X 0,Y 601.417,Z 346.567,A -85,B 0,C 180,E1 -567.868,E2 -567.868} C_VEL
LIN {X 0,Y 601.421,Z 346.572,A -85,B 0,C 180,E1 -570.165,E2 -570.165} C_VEL
LIN {X 0,Y 601.423,Z 346.566,A -85,B 0,C 180,E1 -572.718,E2 -572.718} C_VEL
LIN {X 0,Y 601.405,Z 346.566,A -85,B 0,C 180,E1 -575.115,E2 -575.115} C_VEL
LIN {X 0,Y 601.432,Z 346.563,A -85,B 0,C 180,E1 -577.42,E2 -577.42} C_VEL
LIN {X 0,Y 601.411,Z 346.574,A -85,B 0,C 180,E1 -579.996,E2 -579.996} C_VEL
LIN {X 0,Y 601.412,Z 346.566,A -85,B 0,C 180,E1 -582.671,E2 -582.671} C_VEL
LIN {X 0,Y 601.423,Z 346.567,A -85,B 0,C 180,E1 -585.483,E2 -585.483} C_VEL
LIN {X 0,Y 601.424,Z 346.566,A -85,B 0,C 180,E1 -588.408,E2 -588.408} C_VEL
LIN {X 0,Y 601.435,Z 346.562,A -85,B 0,C 180,E1 -590.876,E2 -590.876} C_VEL
LIN {X 0,Y 601.445,Z 346.571,A -85,B 0,C 180,E1 -593.735,E2 -593.735} C_VEL
LIN {X 0,Y 601.434,Z 346.567,A -85,B 0,C 180,E1 -596.065,E2 -596.065} C_VEL
LIN {X 0,Y 601.422,Z 346.564,A -85,B 0,C 180,E1 -598.546,E2 -598.546} C_VEL
LIN {X 0,Y 601.445,Z 346.565,A -85,B 0,C 180,E1 -601.211,E2 -601.211} C_VEL
LIN {X 0,Y 601.439,Z 346.646,A -85,B 0,C 180,E1 -602.913,E2 -602.913} C_VEL
LIN {X 0,Y 601.427,Z 360.858,A -85,B 0,C 180,E1 -605.453,E2 -605.453} C_VEL
LIN {X 0,Y 601.417,Z 374.632,A -85,B 0,C 180,E1 -607.886,E2 -607.886} C_VEL
LIN {X 0,Y 601.681,Z 380.134,A -85,B 0,C 180,E1 -607.963,E2 -607.963} C_VEL
LIN {X 0,Y 601.596,Z 481.162,A -85,B 0,C 180,E1 -609.188,E2 -609.188} C_VEL
LIN {X 0,Y 601.556,Z 494.239,A -85,B 0,C 180,E1 -609.483,E2 -609.483} C_VEL
LIN {X 0,Y 601.559,Z 507.448,A -85,B 0,C 180,E1 -609.929,E2 -609.929} C_VEL
LIN {X 0,Y 601.515,Z 519.014,A -85,B 0,C 180,E1 -610.461,E2 -610.461} C_VEL
LIN {X 0,Y 601.446,Z 531.023,A -85,B 0,C 180,E1 -611.175,E2 -611.175} C_VEL
LIN {X 0,Y 601.469,Z 541.569,A -85,B 0,C 180,E1 -611.963,E2 -611.963} C_VEL
LIN {X 0,Y 601.396,Z 551.017,A -85,B 0,C 180,E1 -612.838,E2 -612.838} C_VEL
LIN {X 0,Y 601.408,Z 560.162,A -85,B 0,C 180,E1 -613.887,E2 -613.887} C_VEL
LIN {X 0,Y 601.371,Z 567.393,A -85,B 0,C 180,E1 -614.929,E2 -614.929} C_VEL
LIN {X 0,Y 601.353,Z 572.982,A -85,B 0,C 180,E1 -615.937,E2 -615.937} C_VEL
LIN {X 0,Y 601.335,Z 578.215,A -85,B 0,C 180,E1 -617.17,E2 -617.17} C_VEL
LIN {X 0,Y 601.368,Z 580.46,A -85,B 0,C 180,E1 -617.857,E2 -617.857} C_VEL
LIN {X 0,Y 601.337,Z 583.2,A -85,B 0,C 180,E1 -619.035,E2 -619.035} C_VEL
LIN {X 0,Y 601.329,Z 584.414,A -85,B 0,C 180,E1 -619.903,E2 -619.903} C_VEL
LIN {X 0,Y 601.335,Z 584.899,A -85,B 0,C 180,E1 -620.583,E2 -620.583} C_VEL
LIN {X 0,Y 601.333,Z 584.629,A -85,B 0,C 180,E1 -621.938,E2 -621.938} C_VEL
LIN {X 0,Y 601.322,Z 583.913,A -85,B 0,C 180,E1 -622.614,E2 -622.614} C_VEL
LIN {X 0,Y 601.35,Z 582.48,A -85,B 0,C 180,E1 -623.417,E2 -623.417} C_VEL
LIN {X 0,Y 601.352,Z 579.198,A -85,B 0,C 180,E1 -624.635,E2 -624.635} C_VEL
LIN {X 0,Y 601.355,Z 575.348,A -85,B 0,C 180,E1 -625.643,E2 -625.643} C_VEL
LIN {X 0,Y 601.353,Z 570.384,A -85,B 0,C 180,E1 -626.65,E2 -626.65} C_VEL
LIN {X 0,Y 601.394,Z 564.164,A -85,B 0,C 180,E1 -627.656,E2 -627.656} C_VEL
LIN {X 0,Y 601.406,Z 556.424,A -85,B 0,C 180,E1 -628.661,E2 -628.661} C_VEL
LIN {X 0,Y 601.415,Z 546.795,A -85,B 0,C 180,E1 -629.665,E2 -629.665} C_VEL
LIN {X 0,Y 601.451,Z 536.844,A -85,B 0,C 180,E1 -630.502,E2 -630.502} C_VEL
LIN {X 0,Y 601.469,Z 525.655,A -85,B 0,C 180,E1 -631.255,E2 -631.255} C_VEL
LIN {X 0,Y 601.498,Z 514.73,A -85,B 0,C 180,E1 -631.841,E2 -631.841} C_VEL
LIN {X 0,Y 601.537,Z 502.633,A -85,B 0,C 180,E1 -632.344,E2 -632.344} C_VEL
LIN {X 0,Y 601.568,Z 489.914,A -85,B 0,C 180,E1 -632.72,E2 -632.72} C_VEL
LIN {X 0,Y 601.594,Z 476.494,A -85,B 0,C 180,E1 -632.971,E2 -632.971} C_VEL
LIN {X 0,Y 601.5,Z 375.411,A -85,B 0,C 180,E1 -634.188,E2 -634.188} C_VEL
LIN {X 0,Y 601.406,Z 374.482,A -85,B 0,C 180,E1 -634.23,E2 -634.23} C_VEL
LIN {X 0,Y 601.467,Z 358.543,A -85,B 0,C 180,E1 -637.047,E2 -637.047} C_VEL
LIN {X 0,Y 601.441,Z 346.564,A -85,B 0,C 180,E1 -639.203,E2 -639.203} C_VEL
LIN {X 0,Y 601.422,Z 346.569,A -85,B 0,C 180,E1 -642.142,E2 -642.142} C_VEL
LIN {X 0,Y 601.434,Z 346.565,A -85,B 0,C 180,E1 -644.896,E2 -644.896} C_VEL
LIN {X 0,Y 601.435,Z 346.563,A -85,B 0,C 180,E1 -646.985,E2 -646.985} C_VEL
LIN {X 0,Y 601.408,Z 346.568,A -85,B 0,C 180,E1 -649.809,E2 -649.809} C_VEL
LIN {X 0,Y 601.42,Z 346.568,A -85,B 0,C 180,E1 -652.605,E2 -652.605} C_VEL
LIN {X 0,Y 601.404,Z 346.567,A -85,B 0,C 180,E1 -654.878,E2 -654.878} C_VEL
LIN {X 0,Y 601.423,Z 346.569,A -85,B 0,C 180,E1 -657.867,E2 -657.867} C_VEL
LIN {X 0,Y 601.452,Z 346.57,A -85,B 0,C 180,E1 -660.162,E2 -660.162} C_VEL
LIN {X 0,Y 601.422,Z 346.565,A -85,B 0,C 180,E1 -662.714,E2 -662.714} C_VEL
LIN {X 0,Y 601.417,Z 346.564,A -85,B 0,C 180,E1 -665.114,E2 -665.114} C_VEL
LIN {X 0,Y 601.434,Z 346.564,A -85,B 0,C 180,E1 -667.418,E2 -667.418} C_VEL
LIN {X 0,Y 601.41,Z 346.575,A -85,B 0,C 180,E1 -669.994,E2 -669.994} C_VEL
LIN {X 0,Y 601.407,Z 346.566,A -85,B 0,C 180,E1 -672.669,E2 -672.669} C_VEL
LIN {X 0,Y 601.423,Z 346.568,A -85,B 0,C 180,E1 -675.481,E2 -675.481} C_VEL
LIN {X 0,Y 601.422,Z 346.565,A -85,B 0,C 180,E1 -678.406,E2 -678.406} C_VEL
LIN {X 0,Y 601.431,Z 346.563,A -85,B 0,C 180,E1 -680.874,E2 -680.874} C_VEL
LIN {X 0,Y 601.438,Z 346.571,A -85,B 0,C 180,E1 -683.733,E2 -683.733} C_VEL
LIN {X 0,Y 601.426,Z 346.563,A -85,B 0,C 180,E1 -686.686,E2 -686.686} C_VEL
LIN {X 0,Y 601.425,Z 346.565,A -85,B 0,C 180,E1 -689.058,E2 -689.058} C_VEL
LIN {X 0,Y 601.435,Z 346.569,A -85,B 0,C 180,E1 -691.373,E2 -691.373} C_VEL
LIN {X 0,Y 601.402,Z 346.574,A -85,B 0,C 180,E1 -693.636,E2 -693.636} C_VEL
LIN {X 0,Y 601.417,Z 346.564,A -85,B 0,C 180,E1 -696.589,E2 -696.589} C_VEL
LIN {X 0,Y 601.432,Z 346.571,A -85,B 0,C 180,E1 -699.478,E2 -699.478} C_VEL
LIN {X 0,Y 601.397,Z 346.567,A -85,B 0,C 180,E1 -702.311,E2 -702.311} C_VEL
LIN {X 0,Y 601.414,Z 346.565,A -85,B 0,C 180,E1 -704.408,E2 -704.408} C_VEL
LIN {X 0,Y 601.425,Z 346.572,A -85,B 0,C 180,E1 -707.172,E2 -707.172} C_VEL
LIN {X 0,Y 601.43,Z 346.563,A -85,B 0,C 180,E1 -709.905,E2 -709.905} C_VEL
LIN {X 0,Y 601.448,Z 346.563,A -85,B 0,C 180,E1 -712.615,E2 -712.615} C_VEL
LIN {X 0,Y 601.429,Z 346.57,A -85,B 0,C 180,E1 -715.308,E2 -715.308} C_VEL
LIN {X 0,Y 601.418,Z 346.564,A -85,B 0,C 180,E1 -717.991,E2 -717.991} C_VEL
LIN {X 0,Y 601.455,Z 346.564,A -85,B 0,C 180,E1 -720.669,E2 -720.669} C_VEL
LIN {X 0,Y 601.433,Z 346.566,A -85,B 0,C 180,E1 -723.349,E2 -723.349} C_VEL
LIN {X 0,Y 601.405,Z 346.566,A -85,B 0,C 180,E1 -726.037,E2 -726.037} C_VEL
LIN {X 0,Y 601.438,Z 346.57,A -85,B 0,C 180,E1 -728.737,E2 -728.737} C_VEL
LIN {X 0,Y 601.43,Z 346.564,A -85,B 0,C 180,E1 -731.458,E2 -731.458} C_VEL
LIN {X 0,Y 601.411,Z 346.567,A -85,B 0,C 180,E1 -734.206,E2 -734.206} C_VEL
LIN {X 0,Y 601.431,Z 346.568,A -85,B 0,C 180,E1 -736.986,E2 -736.986} C_VEL
LIN {X 0,Y 601.404,Z 346.566,A -85,B 0,C 180,E1 -739.809,E2 -739.809} C_VEL
LIN {X 0,Y 601.448,Z 346.569,A -85,B 0,C 180,E1 -742.682,E2 -742.682} C_VEL
LIN {X 0,Y 601.4,Z 346.571,A -85,B 0,C 180,E1 -744.879,E2 -744.879} C_VEL
LIN {X 0,Y 601.419,Z 346.565,A -85,B 0,C 180,E1 -747.867,E2 -747.867} C_VEL
LIN {X 0,Y 601.42,Z 346.569,A -85,B 0,C 180,E1 -750.165,E2 -750.165} C_VEL
LIN {X 0,Y 601.426,Z 346.568,A -85,B 0,C 180,E1 -752.718,E2 -752.718} C_VEL
LIN {X 0,Y 601.405,Z 346.566,A -85,B 0,C 180,E1 -755.115,E2 -755.115} C_VEL
LIN {X 0,Y 601.43,Z 346.562,A -85,B 0,C 180,E1 -757.419,E2 -757.419} C_VEL
LIN {X 0,Y 601.406,Z 346.571,A -85,B 0,C 180,E1 -759.996,E2 -759.996} C_VEL
LIN {X 0,Y 601.411,Z 346.568,A -85,B 0,C 180,E1 -762.67,E2 -762.67} C_VEL
LIN {X 0,Y 601.421,Z 346.564,A -85,B 0,C 180,E1 -765.483,E2 -765.483} C_VEL
LIN {X 0,Y 601.421,Z 346.569,A -85,B 0,C 180,E1 -768.407,E2 -768.407} C_VEL
LIN {X 0,Y 601.434,Z 346.562,A -85,B 0,C 180,E1 -770.876,E2 -770.876} C_VEL
LIN {X 0,Y 601.442,Z 346.566,A -85,B 0,C 180,E1 -773.734,E2 -773.734} C_VEL
LIN {X 0,Y 601.433,Z 346.571,A -85,B 0,C 180,E1 -776.065,E2 -776.065} C_VEL
LIN {X 0,Y 601.441,Z 346.563,A -85,B 0,C 180,E1 -778.543,E2 -778.543} C_VEL
LIN {X 0,Y 601.433,Z 346.565,A -85,B 0,C 180,E1 -781.374,E2 -781.374} C_VEL
LIN {X 0,Y 601.414,Z 346.57,A -85,B 0,C 180,E1 -784.133,E2 -784.133} C_VEL
LIN {X 0,Y 601.427,Z 346.655,A -85,B 0,C 180,E1 -786.75,E2 -786.75} C_VEL
LIN {X 0,Y 601.715,Z 351.666,A -85,B 0,C 180,E1 -787.446,E2 -787.446} C_VEL
LIN {X 0,Y 601.599,Z 372.083,A -85,B 0,C 180,E1 -790.198,E2 -790.198} C_VEL
LIN {X 0,Y 601.547,Z 393.356,A -85,B 0,C 180,E1 -793.018,E2 -793.018} C_VEL
LIN {X 0,Y 601.504,Z 416.28,A -85,B 0,C 180,E1 -796.011,E2 -796.011} C_VEL
LIN {X 0,Y 601.469,Z 422.524,A -85,B 0,C 180,E1 -796.819,E2 -796.819} C_VEL
LIN {X 0,Y 601.662,Z 439.266,A -85,B 0,C 180,E1 -797.027,E2 -797.027} C_VEL
LIN {X 0,Y 601.605,Z 530.962,A -85,B 0,C 180,E1 -798.14,E2 -798.14} C_VEL
LIN {X 0,Y 601.574,Z 544.227,A -85,B 0,C 180,E1 -798.438,E2 -798.438} C_VEL
LIN {X 0,Y 601.54,Z 556.706,A -85,B 0,C 180,E1 -798.856,E2 -798.856} C_VEL
LIN {X 0,Y 601.523,Z 568.638,A -85,B 0,C 180,E1 -799.396,E2 -799.396} C_VEL
LIN {X 0,Y 601.481,Z 580.202,A -85,B 0,C 180,E1 -800.076,E2 -800.076} C_VEL
LIN {X 0,Y 601.444,Z 590.598,A -85,B 0,C 180,E1 -800.839,E2 -800.839} C_VEL
LIN {X 0,Y 601.429,Z 599.114,A -85,B 0,C 180,E1 -801.601,E2 -801.601} C_VEL
LIN {X 0,Y 601.418,Z 606.962,A -85,B 0,C 180,E1 -802.446,E2 -802.446} C_VEL
LIN {X 0,Y 601.37,Z 614.225,A -85,B 0,C 180,E1 -803.398,E2 -803.398} C_VEL
LIN {X 0,Y 601.372,Z 619.867,A -85,B 0,C 180,E1 -804.299,E2 -804.299} C_VEL
LIN {X 0,Y 601.337,Z 624.95,A -85,B 0,C 180,E1 -805.307,E2 -805.307} C_VEL
LIN {X 0,Y 601.367,Z 628.896,A -85,B 0,C 180,E1 -806.315,E2 -806.315} C_VEL
LIN {X 0,Y 601.325,Z 631.809,A -85,B 0,C 180,E1 -807.321,E2 -807.321} C_VEL
LIN {X 0,Y 601.341,Z 633.202,A -85,B 0,C 180,E1 -807.991,E2 -807.991} C_VEL
LIN {X 0,Y 601.339,Z 634.784,A -85,B 0,C 180,E1 -809.33,E2 -809.33} C_VEL
LIN {X 0,Y 601.335,Z 635,A -85,B 0,C 180,E1 -810,E2 -810} C_VEL
LIN {X 0,Y 601.348,Z 634.184,A -85,B 0,C 180,E1 -811.339,E2 -811.339} C_VEL
LIN {X 0,Y 601.341,Z 633.202,A -85,B 0,C 180,E1 -812.009,E2 -812.009} C_VEL
LIN {X 0,Y 601.325,Z 631.809,A -85,B 0,C 180,E1 -812.679,E2 -812.679} C_VEL
LIN {X 0,Y 601.367,Z 628.896,A -85,B 0,C 180,E1 -813.685,E2 -813.685} C_VEL
LIN {X 0,Y 601.337,Z 624.95,A -85,B 0,C 180,E1 -814.693,E2 -814.693} C_VEL
LIN {X 0,Y 601.372,Z 618.878,A -85,B 0,C 180,E1 -815.869,E2 -815.869} C_VEL
LIN {X 0,Y 601.381,Z 612.237,A -85,B 0,C 180,E1 -816.88,E2 -816.88} C_VEL
LIN {X 0,Y 601.4,Z 603.991,A -85,B 0,C 180,E1 -817.892,E2 -817.892} C_VEL
LIN {X 0,Y 601.436,Z 595.539,A -85,B 0,C 180,E1 -818.737,E2 -818.737} C_VEL
LIN {X 0,Y 601.442,Z 585.095,A -85,B 0,C 180,E1 -819.585,E2 -819.585} C_VEL
LIN {X 0,Y 601.472,Z 574.761,A -85,B 0,C 180,E1 -820.264,E2 -820.264} C_VEL
LIN {X 0,Y 601.536,Z 563.907,A -85,B 0,C 180,E1 -820.835,E2 -820.835} C_VEL
LIN {X 0,Y 601.556,Z 551.385,A -85,B 0,C 180,E1 -821.34,E2 -821.34} C_VEL
LIN {X 0,Y 601.568,Z 538.363,A -85,B 0,C 180,E1 -821.711,E2 -821.711} C_VEL
LIN {X 0,Y 601.614,Z 525.105,A -85,B 0,C 180,E1 -821.946,E2 -821.946} C_VEL
LIN {X 0,Y 601.548,Z 423.168,A -85,B 0,C 180,E1 -823.169,E2 -823.169} C_VEL
LIN {X 0,Y 601.467,Z 422.275,A -85,B 0,C 180,E1 -823.213,E2 -823.213} C_VEL
LIN {X 0,Y 601.52,Z 400.004,A -85,B 0,C 180,E1 -826.11,E2 -826.11} C_VEL
LIN {X 0,Y 601.606,Z 377.402,A -85,B 0,C 180,E1 -829.092,E2 -829.092} C_VEL
LIN {X 0,Y 601.677,Z 356.128,A -85,B 0,C 180,E1 -831.948,E2 -831.948} C_VEL
LIN {X 0,Y 601.69,Z 348.151,A -85,B 0,C 180,E1 -833.034,E2 -833.034} C_VEL
LIN {X 0,Y 601.414,Z 346.569,A -85,B 0,C 180,E1 -833.273,E2 -833.273} C_VEL
LIN {X 0,Y 601.414,Z 346.57,A -85,B 0,C 180,E1 -835.867,E2 -835.867} C_VEL
LIN {X 0,Y 601.433,Z 346.564,A -85,B 0,C 180,E1 -838.626,E2 -838.626} C_VEL
LIN {X 0,Y 601.441,Z 346.563,A -85,B 0,C 180,E1 -841.458,E2 -841.458} C_VEL
LIN {X 0,Y 601.431,Z 346.571,A -85,B 0,C 180,E1 -844.117,E2 -844.117} C_VEL
LIN {X 0,Y 601.411,Z 346.566,A -85,B 0,C 180,E1 -846.581,E2 -846.581} C_VEL
LIN {X 0,Y 601.44,Z 346.566,A -85,B 0,C 180,E1 -849.535,E2 -849.535} C_VEL
LIN {X 0,Y 601.407,Z 346.566,A -85,B 0,C 180,E1 -852.59,E2 -852.59} C_VEL
LIN {X 0,Y 601.421,Z 346.569,A -85,B 0,C 180,E1 -855.481,E2 -855.481} C_VEL
LIN {X 0,Y 601.422,Z 346.564,A -85,B 0,C 180,E1 -858.406,E2 -858.406} C_VEL
LIN {X 0,Y 601.431,Z 346.563,A -85,B 0,C 180,E1 -860.875,E2 -860.875} C_VEL
LIN {X 0,Y 601.438,Z 346.569,A -85,B 0,C 180,E1 -863.733,E2 -863.733} C_VEL
LIN {X 0,Y 601.426,Z 346.563,A -85,B 0,C 180,E1 -866.686,E2 -866.686} C_VEL
LIN {X 0,Y 601.426,Z 346.566,A -85,B 0,C 180,E1 -869.058,E2 -869.058} C_VEL
LIN {X 0,Y 601.436,Z 346.571,A -85,B 0,C 180,E1 -871.373,E2 -871.373} C_VEL
LIN {X 0,Y 601.403,Z 346.571,A -85,B 0,C 180,E1 -873.636,E2 -873.636} C_VEL
LIN {X 0,Y 601.418,Z 346.564,A -85,B 0,C 180,E1 -876.59,E2 -876.59} C_VEL
LIN {X 0,Y 601.433,Z 346.569,A -85,B 0,C 180,E1 -879.478,E2 -879.478} C_VEL
LIN {X 0,Y 601.398,Z 346.566,A -85,B 0,C 180,E1 -882.312,E2 -882.312} C_VEL
LIN {X 0,Y 601.414,Z 346.565,A -85,B 0,C 180,E1 -884.409,E2 -884.409} C_VEL
LIN {X 0,Y 601.425,Z 346.573,A -85,B 0,C 180,E1 -887.172,E2 -887.172} C_VEL
LIN {X 0,Y 601.43,Z 346.562,A -85,B 0,C 180,E1 -889.905,E2 -889.905} C_VEL
LIN {X 0,Y 601.45,Z 346.564,A -85,B 0,C 180,E1 -892.615,E2 -892.615} C_VEL
LIN {X 0,Y 601.428,Z 346.567,A -85,B 0,C 180,E1 -895.308,E2 -895.308} C_VEL
LIN {X 0,Y 601.418,Z 346.564,A -85,B 0,C 180,E1 -897.991,E2 -897.991} C_VEL
LIN {X 0,Y 601.457,Z 346.566,A -85,B 0,C 180,E1 -900.67,E2 -900.67} C_VEL
LIN {X 0,Y 601.433,Z 346.564,A -85,B 0,C 180,E1 -903.35,E2 -903.35} C_VEL
LIN {X 0,Y 601.405,Z 346.566,A -85,B 0,C 180,E1 -906.037,E2 -906.037} C_VEL
LIN {X 0,Y 601.439,Z 346.571,A -85,B 0,C 180,E1 -908.738,E2 -908.738} C_VEL
LIN {X 0,Y 601.429,Z 346.563,A -85,B 0,C 180,E1 -911.458,E2 -911.458} C_VEL
LIN {X 0,Y 601.408,Z 346.568,A -85,B 0,C 180,E1 -912.393,E2 -912.393} C_VEL
LIN {X 0,Y 600.748,Z 346.653,A -85,B 0,C 180,E1 -912.952,E2 -912.952} C_VEL
LIN {X 0,Y 597.898,Z 347.008,A -85,B 0,C 180,E1 -913.86,E2 -913.86} C_VEL
LIN {X 0,Y 595.484,Z 347.313,A -85,B 0,C 180,E1 -914.59,E2 -914.59} C_VEL
LIN {X 0,Y 594.444,Z 347.435,A -85,B 0,C 180,E1 -915.154,E2 -915.154} C_VEL
LIN {X 0,Y 594.359,Z 347.444,A -85,B 0,C 180,E1 -915.345,E2 -915.345} C_VEL
LIN {X 0,Y 594.374,Z 347.443,A -85,B 0,C 180,E1 -917.905,E2 -917.905} C_VEL
LIN {X 0,Y 594.377,Z 347.444,A -85,B 0,C 180,E1 -920.919,E2 -920.919} C_VEL
LIN {X 0,Y 594.384,Z 347.441,A -85,B 0,C 180,E1 -923.705,E2 -923.705} C_VEL
LIN {X 0,Y 594.381,Z 347.444,A -85,B 0,C 180,E1 -926.7,E2 -926.7} C_VEL
LIN {X 0,Y 594.376,Z 347.442,A -85,B 0,C 180,E1 -928.999,E2 -928.999} C_VEL
LIN {X 0,Y 594.388,Z 347.441,A -85,B 0,C 180,E1 -931.646,E2 -931.646} C_VEL
LIN {X 0,Y 594.387,Z 347.443,A -85,B 0,C 180,E1 -934.58,E2 -934.58} C_VEL
LIN {X 0,Y 594.382,Z 347.44,A -85,B 0,C 180,E1 -937.087,E2 -937.087} C_VEL
LIN {X 0,Y 594.374,Z 347.447,A -85,B 0,C 180,E1 -939.776,E2 -939.776} C_VEL
LIN {X 0,Y 594.371,Z 347.446,A -85,B 0,C 180,E1 -942.376,E2 -942.376} C_VEL
LIN {X 0,Y 594.361,Z 347.444,A -85,B 0,C 180,E1 -945.192,E2 -945.192} C_VEL
LIN {X 0,Y 594.37,Z 347.448,A -85,B 0,C 180,E1 -947.626,E2 -947.626} C_VEL
LIN {X 0,Y 594.394,Z 347.442,A -85,B 0,C 180,E1 -950.322,E2 -950.322} C_VEL
LIN {X 0,Y 594.386,Z 347.44,A -85,B 0,C 180,E1 -952.914,E2 -952.914} C_VEL
LIN {X 0,Y 594.387,Z 347.448,A -85,B 0,C 180,E1 -955.862,E2 -955.862} C_VEL
LIN {X 0,Y 594.373,Z 347.442,A -85,B 0,C 180,E1 -958.651,E2 -958.651} C_VEL
LIN {X 0,Y 594.388,Z 347.442,A -85,B 0,C 180,E1 -961.043,E2 -961.043} C_VEL
LIN {X 0,Y 594.409,Z 347.528,A -85,B 0,C 180,E1 -962.851,E2 -962.851} C_VEL
LIN {X 0,Y 594.412,Z 360.404,A -85,B 0,C 180,E1 -965.183,E2 -965.183} C_VEL
LIN {X 0,Y 594.35,Z 374.601,A -85,B 0,C 180,E1 -967.721,E2 -967.721} C_VEL
LIN {X 0,Y 594.777,Z 379.955,A -85,B 0,C 180,E1 -967.806,E2 -967.806} C_VEL
LIN {X 0,Y 594.666,Z 481.572,A -85,B 0,C 180,E1 -969.056,E2 -969.056} C_VEL
LIN {X 0,Y 594.616,Z 494.221,A -85,B 0,C 180,E1 -969.346,E2 -969.346} C_VEL
LIN {X 0,Y 594.6,Z 506.846,A -85,B 0,C 180,E1 -969.774,E2 -969.774} C_VEL
LIN {X 0,Y 594.527,Z 518.583,A -85,B 0,C 180,E1 -970.312,E2 -970.312} C_VEL
LIN {X 0,Y 594.45,Z 529.957,A -85,B 0,C 180,E1 -970.986,E2 -970.986} C_VEL
LIN {X 0,Y 594.424,Z 541.284,A -85,B 0,C 180,E1 -971.83,E2 -971.83} C_VEL
LIN {X 0,Y 594.37,Z 549.956,A -85,B 0,C 180,E1 -972.629,E2 -972.629} C_VEL
LIN {X 0,Y 594.315,Z 559.275,A -85,B 0,C 180,E1 -973.689,E2 -973.689} C_VEL
LIN {X 0,Y 594.307,Z 566.724,A -85,B 0,C 180,E1 -974.745,E2 -974.745} C_VEL
LIN {X 0,Y 594.265,Z 572.985,A -85,B 0,C 180,E1 -975.876,E2 -975.876} C_VEL
LIN {X 0,Y 594.26,Z 577.819,A -85,B 0,C 180,E1 -977.015,E2 -977.015} C_VEL
LIN {X 0,Y 594.258,Z 580.126,A -85,B 0,C 180,E1 -977.709,E2 -977.709} C_VEL
LIN {X 0,Y 594.252,Z 583.178,A -85,B 0,C 180,E1 -978.998,E2 -978.998} C_VEL
LIN {X 0,Y 594.23,Z 584.291,A -85,B 0,C 180,E1 -979.782,E2 -979.782} C_VEL
LIN {X 0,Y 594.255,Z 584.854,A -85,B 0,C 180,E1 -980.47,E2 -980.47} C_VEL
LIN {X 0,Y 594.227,Z 584.981,A -85,B 0,C 180,E1 -981.156,E2 -981.156} C_VEL
LIN {X 0,Y 594.247,Z 584.041,A -85,B 0,C 180,E1 -982.525,E2 -982.525} C_VEL
LIN {X 0,Y 594.264,Z 582.521,A -85,B 0,C 180,E1 -983.426,E2 -983.426} C_VEL
LIN {X 0,Y 594.266,Z 579.532,A -85,B 0,C 180,E1 -984.571,E2 -984.571} C_VEL
LIN {X 0,Y 594.271,Z 575.796,A -85,B 0,C 180,E1 -985.591,E2 -985.591} C_VEL
LIN {X 0,Y 594.275,Z 570.954,A -85,B 0,C 180,E1 -986.61,E2 -986.61} C_VEL
LIN {X 0,Y 594.303,Z 564.869,A -85,B 0,C 180,E1 -987.628,E2 -987.628} C_VEL
LIN {X 0,Y 594.34,Z 557.329,A -85,B 0,C 180,E1 -988.645,E2 -988.645} C_VEL
LIN {X 0,Y 594.366,Z 549.653,A -85,B 0,C 180,E1 -989.492,E2 -989.492} C_VEL
LIN {X 0,Y 594.42,Z 539.262,A -85,B 0,C 180,E1 -990.423,E2 -990.423} C_VEL
LIN {X 0,Y 594.447,Z 528.742,A -85,B 0,C 180,E1 -991.185,E2 -991.185} C_VEL
LIN {X 0,Y 594.484,Z 518.588,A -85,B 0,C 180,E1 -991.778,E2 -991.778} C_VEL
LIN {X 0,Y 594.555,Z 506.531,A -85,B 0,C 180,E1 -992.329,E2 -992.329} C_VEL
LIN {X 0,Y 594.609,Z 493.203,A -85,B 0,C 180,E1 -992.773,E2 -992.773} C_VEL
LIN {X 0,Y 594.638,Z 480.838,A -85,B 0,C 180,E1 -993.049,E2 -993.049} C_VEL
LIN {X 0,Y 594.64,Z 376.493,A -85,B 0,C 180,E1 -994.329,E2 -994.329} C_VEL
LIN {X 0,Y 594.358,Z 374.617,A -85,B 0,C 180,E1 -994.365,E2 -994.365} C_VEL
LIN {X 0,Y 594.442,Z 359.157,A -85,B 0,C 180,E1 -997.131,E2 -997.131} C_VEL
LIN {X 0,Y 594.414,Z 347.44,A -85,B 0,C 180,E1 -999.27,E2 -999.27} C_VEL
LIN {X 0,Y 594.396,Z 347.447,A -85,B 0,C 180,E1 -1002.288,E2 -1002.288} C_VEL
LIN {X 0,Y 594.377,Z 347.442,A -85,B 0,C 180,E1 -1005.077,E2 -1005.077} C_VEL
LIN {X 0,Y 594.393,Z 347.439,A -85,B 0,C 180,E1 -1007.193,E2 -1007.193} C_VEL
LIN {X 0,Y 594.379,Z 347.447,A -85,B 0,C 180,E1 -1010.053,E2 -1010.053} C_VEL
LIN {X 0,Y 594.368,Z 347.443,A -85,B 0,C 180,E1 -1012.967,E2 -1012.967} C_VEL
LIN {X 0,Y 594.377,Z 347.441,A -85,B 0,C 180,E1 -1015.192,E2 -1015.192} C_VEL
LIN {X 0,Y 594.389,Z 347.441,A -85,B 0,C 180,E1 -1017.526,E2 -1017.526} C_VEL
LIN {X 0,Y 594.402,Z 347.445,A -85,B 0,C 180,E1 -1020.33,E2 -1020.33} C_VEL
LIN {X 0,Y 594.379,Z 347.441,A -85,B 0,C 180,E1 -1022.949,E2 -1022.949} C_VEL
LIN {X 0,Y 594.385,Z 347.442,A -85,B 0,C 180,E1 -1025.406,E2 -1025.406} C_VEL
LIN {X 0,Y 594.388,Z 347.45,A -85,B 0,C 180,E1 -1027.94,E2 -1027.94} C_VEL
LIN {X 0,Y 594.374,Z 347.442,A -85,B 0,C 180,E1 -1030.821,E2 -1030.821} C_VEL
LIN {X 0,Y 594.364,Z 347.445,A -85,B 0,C 180,E1 -1033.299,E2 -1033.299} C_VEL
LIN {X 0,Y 594.38,Z 347.445,A -85,B 0,C 180,E1 -1036.158,E2 -1036.158} C_VEL
LIN {X 0,Y 594.375,Z 347.443,A -85,B 0,C 180,E1 -1039.177,E2 -1039.177} C_VEL
LIN {X 0,Y 594.384,Z 347.445,A -85,B 0,C 180,E1 -1042.059,E2 -1042.059} C_VEL
LIN {X 0,Y 594.35,Z 347.445,A -85,B 0,C 180,E1 -1044.675,E2 -1044.675} C_VEL
LIN {X 0,Y 594.376,Z 347.444,A -85,B 0,C 180,E1 -1047.087,E2 -1047.087} C_VEL
LIN {X 0,Y 594.381,Z 347.45,A -85,B 0,C 180,E1 -1049.671,E2 -1049.671} C_VEL
LIN {X 0,Y 594.366,Z 347.443,A -85,B 0,C 180,E1 -1052.538,E2 -1052.538} C_VEL
LIN {X 0,Y 594.372,Z 347.443,A -85,B 0,C 180,E1 -1054.806,E2 -1054.806} C_VEL
LIN {X 0,Y 594.397,Z 347.446,A -85,B 0,C 180,E1 -1057.254,E2 -1057.254} C_VEL
LIN {X 0,Y 594.374,Z 347.444,A -85,B 0,C 180,E1 -1059.946,E2 -1059.946} C_VEL
LIN {X 0,Y 594.388,Z 347.442,A -85,B 0,C 180,E1 -1062.806,E2 -1062.806} C_VEL
LIN {X 0,Y 594.38,Z 347.443,A -85,B 0,C 180,E1 -1065.825,E2 -1065.825} C_VEL
LIN {X 0,Y 594.388,Z 347.44,A -85,B 0,C 180,E1 -1068.404,E2 -1068.404} C_VEL
LIN {X 0,Y 594.398,Z 347.449,A -85,B 0,C 180,E1 -1071.158,E2 -1071.158} C_VEL
LIN {X 0,Y 594.398,Z 347.446,A -85,B 0,C 180,E1 -1073.299,E2 -1073.299} C_VEL
LIN {X 0,Y 594.355,Z 347.444,A -85,B 0,C 180,E1 -1075.931,E2 -1075.931} C_VEL
LIN {X 0,Y 594.389,Z 347.44,A -85,B 0,C 180,E1 -1077.967,E2 -1077.967} C_VEL
LIN {X 0,Y 594.425,Z 347.44,A -85,B 0,C 180,E1 -1080.677,E2 -1080.677} C_VEL
LIN {X 0,Y 594.384,Z 347.444,A -85,B 0,C 180,E1 -1083.389,E2 -1083.389} C_VEL
LIN {X 0,Y 594.361,Z 347.444,A -85,B 0,C 180,E1 -1086.109,E2 -1086.109} C_VEL
LIN {X 0,Y 594.411,Z 347.438,A -85,B 0,C 180,E1 -1088.157,E2 -1088.157} C_VEL
LIN {X 0,Y 594.39,Z 347.445,A -85,B 0,C 180,E1 -1091.08,E2 -1091.08} C_VEL
LIN {X 0,Y 594.377,Z 347.441,A -85,B 0,C 180,E1 -1093.679,E2 -1093.679} C_VEL
LIN {X 0,Y 594.394,Z 347.449,A -85,B 0,C 180,E1 -1096.723,E2 -1096.723} C_VEL
LIN {X 0,Y 594.364,Z 347.444,A -85,B 0,C 180,E1 -1099.334,E2 -1099.334} C_VEL
LIN {X 0,Y 594.365,Z 347.443,A -85,B 0,C 180,E1 -1101.503,E2 -1101.503} C_VEL
LIN {X 0,Y 594.386,Z 347.44,A -85,B 0,C 180,E1 -1103.704,E2 -1103.704} C_VEL
LIN {X 0,Y 594.383,Z 347.448,A -85,B 0,C 180,E1 -1106.7,E2 -1106.7} C_VEL
LIN {X 0,Y 594.379,Z 347.443,A -85,B 0,C 180,E1 -1108.999,E2 -1108.999} C_VEL
LIN {X 0,Y 594.388,Z 347.44,A -85,B 0,C 180,E1 -1111.646,E2 -1111.646} C_VEL
LIN {X 0,Y 594.388,Z 347.447,A -85,B 0,C 180,E1 -1114.58,E2 -1114.58} C_VEL
LIN {X 0,Y 594.38,Z 347.441,A -85,B 0,C 180,E1 -1117.087,E2 -1117.087} C_VEL
LIN {X 0,Y 594.369,Z 347.445,A -85,B 0,C 180,E1 -1119.775,E2 -1119.775} C_VEL
LIN {X 0,Y 594.368,Z 347.45,A -85,B 0,C 180,E1 -1122.376,E2 -1122.376} C_VEL
LIN {X 0,Y 594.358,Z 347.443,A -85,B 0,C 180,E1 -1125.192,E2 -1125.192} C_VEL
LIN {X 0,Y 594.38,Z 347.451,A -85,B 0,C 180,E1 -1128.152,E2 -1128.152} C_VEL
LIN {X 0,Y 594.386,Z 347.44,A -85,B 0,C 180,E1 -1131.196,E2 -1131.196} C_VEL
LIN {X 0,Y 594.395,Z 347.445,A -85,B 0,C 180,E1 -1133.76,E2 -1133.76} C_VEL
LIN {X 0,Y 594.379,Z 347.447,A -85,B 0,C 180,E1 -1136.24,E2 -1136.24} C_VEL
LIN {X 0,Y 594.39,Z 347.44,A -85,B 0,C 180,E1 -1138.652,E2 -1138.652} C_VEL
LIN {X 0,Y 594.384,Z 347.441,A -85,B 0,C 180,E1 -1141.043,E2 -1141.043} C_VEL
LIN {X 0,Y 594.388,Z 347.449,A -85,B 0,C 180,E1 -1143.977,E2 -1143.977} C_VEL
LIN {X 0,Y 594.393,Z 347.486,A -85,B 0,C 180,E1 -1146.574,E2 -1146.574} C_VEL
LIN {X 0,Y 594.802,Z 351.635,A -85,B 0,C 180,E1 -1147.165,E2 -1147.165} C_VEL
LIN {X 0,Y 594.67,Z 372.083,A -85,B 0,C 180,E1 -1149.957,E2 -1149.957} C_VEL
LIN {X 0,Y 594.572,Z 392.027,A -85,B 0,C 180,E1 -1152.635,E2 -1152.635} C_VEL
LIN {X 0,Y 594.484,Z 414.63,A -85,B 0,C 180,E1 -1155.626,E2 -1155.626} C_VEL
LIN {X 0,Y 594.46,Z 422.524,A -85,B 0,C 180,E1 -1156.661,E2 -1156.661} C_VEL
LIN {X 0,Y 594.783,Z 428.534,A -85,B 0,C 180,E1 -1156.744,E2 -1156.744} C_VEL
LIN {X 0,Y 594.684,Z 530.961,A -85,B 0,C 180,E1 -1158,E2 -1158} C_VEL
LIN {X 0,Y 594.616,Z 544.227,A -85,B 0,C 180,E1 -1158.301,E2 -1158.301} C_VEL
LIN {X 0,Y 594.569,Z 557.413,A -85,B 0,C 180,E1 -1158.75,E2 -1158.75} C_VEL
LIN {X 0,Y 594.537,Z 568.637,A -85,B 0,C 180,E1 -1159.27,E2 -1159.27} C_VEL
LIN {X 0,Y 594.469,Z 580.203,A -85,B 0,C 180,E1 -1159.958,E2 -1159.958} C_VEL
LIN {X 0,Y 594.413,Z 590.599,A -85,B 0,C 180,E1 -1160.73,E2 -1160.73} C_VEL
LIN {X 0,Y 594.383,Z 599.114,A -85,B 0,C 180,E1 -1161.501,E2 -1161.501} C_VEL
LIN {X 0,Y 594.347,Z 606.962,A -85,B 0,C 180,E1 -1162.356,E2 -1162.356} C_VEL
LIN {X 0,Y 594.282,Z 614.813,A -85,B 0,C 180,E1 -1163.408,E2 -1163.408} C_VEL
LIN {X 0,Y 594.289,Z 621.681,A -85,B 0,C 180,E1 -1164.571,E2 -1164.571} C_VEL
LIN {X 0,Y 594.27,Z 626.372,A -85,B 0,C 180,E1 -1165.591,E2 -1165.591} C_VEL
LIN {X 0,Y 594.267,Z 629.957,A -85,B 0,C 180,E1 -1166.61,E2 -1166.61} C_VEL
LIN {X 0,Y 594.226,Z 631.809,A -85,B 0,C 180,E1 -1167.288,E2 -1167.288} C_VEL
LIN {X 0,Y 594.24,Z 633.201,A -85,B 0,C 180,E1 -1167.967,E2 -1167.967} C_VEL
LIN {X 0,Y 594.239,Z 634.784,A -85,B 0,C 180,E1 -1169.322,E2 -1169.322} C_VEL
LIN {X 0,Y 594.236,Z 635,A -85,B 0,C 180,E1 -1170,E2 -1170} C_VEL
LIN {X 0,Y 594.247,Z 634.185,A -85,B 0,C 180,E1 -1171.355,E2 -1171.355} C_VEL
LIN {X 0,Y 594.24,Z 633.202,A -85,B 0,C 180,E1 -1172.033,E2 -1172.033} C_VEL
LIN {X 0,Y 594.226,Z 631.81,A -85,B 0,C 180,E1 -1172.712,E2 -1172.712} C_VEL
LIN {X 0,Y 594.288,Z 628.896,A -85,B 0,C 180,E1 -1173.729,E2 -1173.729} C_VEL
LIN {X 0,Y 594.242,Z 624.95,A -85,B 0,C 180,E1 -1174.749,E2 -1174.749} C_VEL
LIN {X 0,Y 594.304,Z 618.878,A -85,B 0,C 180,E1 -1175.939,E2 -1175.939} C_VEL
LIN {X 0,Y 594.308,Z 612.237,A -85,B 0,C 180,E1 -1176.962,E2 -1176.962} C_VEL
LIN {X 0,Y 594.359,Z 603.991,A -85,B 0,C 180,E1 -1177.986,E2 -1177.986} C_VEL
LIN {X 0,Y 594.382,Z 595.539,A -85,B 0,C 180,E1 -1178.842,E2 -1178.842} C_VEL
LIN {X 0,Y 594.427,Z 585.097,A -85,B 0,C 180,E1 -1179.699,E2 -1179.699} C_VEL
LIN {X 0,Y 594.482,Z 574.763,A -85,B 0,C 180,E1 -1180.386,E2 -1180.386} C_VEL
LIN {X 0,Y 594.559,Z 563.705,A -85,B 0,C 180,E1 -1180.974,E2 -1180.974} C_VEL
LIN {X 0,Y 594.582,Z 551.712,A -85,B 0,C 180,E1 -1181.464,E2 -1181.464} C_VEL
LIN {X 0,Y 594.637,Z 538.363,A -85,B 0,C 180,E1 -1181.85,E2 -1181.85} C_VEL
LIN {X 0,Y 594.693,Z 525.105,A -85,B 0,C 180,E1 -1182.087,E2 -1182.087} C_VEL
LIN {X 0,Y 594.652,Z 423.95,A -85,B 0,C 180,E1 -1183.315,E2 -1183.315} C_VEL
LIN {X 0,Y 594.448,Z 422.441,A -85,B 0,C 180,E1 -1183.35,E2 -1183.35} C_VEL
LIN {X 0,Y 594.533,Z 400.004,A -85,B 0,C 180,E1 -1186.305,E2 -1186.305} C_VEL
LIN {X 0,Y 594.67,Z 377.402,A -85,B 0,C 180,E1 -1189.324,E2 -1189.324} C_VEL
LIN {X 0,Y 594.807,Z 355.013,A -85,B 0,C 180,E1 -1192.369,E2 -1192.369} C_VEL
LIN {X 0,Y 594.758,Z 349.48,A -85,B 0,C 180,E1 -1193.135,E2 -1193.135} C_VEL
LIN {X 0,Y 594.38,Z 347.447,A -85,B 0,C 180,E1 -1193.45,E2 -1193.45} C_VEL
LIN {X 0,Y 594.388,Z 347.449,A -85,B 0,C 180,E1 -1196.023,E2 -1196.023} C_VEL
LIN {X 0,Y 594.384,Z 347.441,A -85,B 0,C 180,E1 -1198.957,E2 -1198.957} C_VEL
LIN {X 0,Y 594.391,Z 347.443,A -85,B 0,C 180,E1 -1201.644,E2 -1201.644} C_VEL
LIN {X 0,Y 594.398,Z 347.44,A -85,B 0,C 180,E1 -1204.578,E2 -1204.578} C_VEL
LIN {X 0,Y 594.383,Z 347.441,A -85,B 0,C 180,E1 -1207.086,E2 -1207.086} C_VEL
LIN {X 0,Y 594.375,Z 347.45,A -85,B 0,C 180,E1 -1209.774,E2 -1209.774} C_VEL
LIN {X 0,Y 594.364,Z 347.445,A -85,B 0,C 180,E1 -1212.375,E2 -1212.375} C_VEL
LIN {X 0,Y 594.358,Z 347.445,A -85,B 0,C 180,E1 -1215.191,E2 -1215.191} C_VEL
LIN {X 0,Y 594.369,Z 347.451,A -85,B 0,C 180,E1 -1217.624,E2 -1217.624} C_VEL
LIN {X 0,Y 594.386,Z 347.441,A -85,B 0,C 180,E1 -1220.32,E2 -1220.32} C_VEL
LIN {X 0,Y 594.381,Z 347.441,A -85,B 0,C 180,E1 -1222.913,E2 -1222.913} C_VEL
LIN {X 0,Y 594.379,Z 347.446,A -85,B 0,C 180,E1 -1225.86,E2 -1225.86} C_VEL
LIN {X 0,Y 594.385,Z 347.44,A -85,B 0,C 180,E1 -1228.651,E2 -1228.651} C_VEL
LIN {X 0,Y 594.382,Z 347.444,A -85,B 0,C 180,E1 -1231.04,E2 -1231.04} C_VEL
LIN {X 0,Y 594.383,Z 347.441,A -85,B 0,C 180,E1 -1233.975,E2 -1233.975} C_VEL
LIN {X 0,Y 594.386,Z 347.439,A -85,B 0,C 180,E1 -1236.296,E2 -1236.296} C_VEL
LIN {X 0,Y 594.406,Z 347.447,A -85,B 0,C 180,E1 -1239.225,E2 -1239.225} C_VEL
LIN {X 0,Y 594.377,Z 347.441,A -85,B 0,C 180,E1 -1242.096,E2 -1242.096} C_VEL
LIN {X 0,Y 594.367,Z 347.442,A -85,B 0,C 180,E1 -1244.219,E2 -1244.219} C_VEL
LIN {X 0,Y 594.371,Z 347.45,A -85,B 0,C 180,E1 -1247.017,E2 -1247.017} C_VEL
LIN {X 0,Y 594.391,Z 347.44,A -85,B 0,C 180,E1 -1249.784,E2 -1249.784} C_VEL
LIN {X 0,Y 594.413,Z 347.439,A -85,B 0,C 180,E1 -1252.527,E2 -1252.527} C_VEL
LIN {X 0,Y 594.396,Z 347.444,A -85,B 0,C 180,E1 -1255.253,E2 -1255.253} C_VEL
LIN {X 0,Y 594.389,Z 347.439,A -85,B 0,C 180,E1 -1257.967,E2 -1257.967} C_VEL
LIN {X 0,Y 594.426,Z 347.442,A -85,B 0,C 180,E1 -1260.678,E2 -1260.678} C_VEL
LIN {X 0,Y 594.383,Z 347.441,A -85,B 0,C 180,E1 -1263.39,E2 -1263.39} C_VEL
LIN {X 0,Y 594.361,Z 347.444,A -85,B 0,C 180,E1 -1266.109,E2 -1266.109} C_VEL
LIN {X 0,Y 594.411,Z 347.439,A -85,B 0,C 180,E1 -1268.157,E2 -1268.157} C_VEL
LIN {X 0,Y 594.389,Z 347.443,A -85,B 0,C 180,E1 -1271.08,E2 -1271.08} C_VEL
LIN {X 0,Y 594.377,Z 347.441,A -85,B 0,C 180,E1 -1273.679,E2 -1273.679} C_VEL
LIN {X 0,Y 594.359,Z 347.444,A -85,B 0,C 180,E1 -1275.345,E2 -1275.345} C_VEL
LIN {X 0,Y 593.688,Z 347.529,A -85,B 0,C 180,E1 -1275.91,E2 -1275.91} C_VEL
LIN {X 0,Y 590.833,Z 347.887,A -85,B 0,C 180,E1 -1276.829,E2 -1276.829} C_VEL
LIN {X 0,Y 588.427,Z 348.187,A -85,B 0,C 180,E1 -1277.567,E2 -1277.567} C_VEL
LIN {X 0,Y 587.399,Z 348.314,A -85,B 0,C 180,E1 -1278.138,E2 -1278.138} C_VEL
LIN {X 0,Y 587.319,Z 348.323,A -85,B 0,C 180,E1 -1278.331,E2 -1278.331} C_VEL
LIN {X 0,Y 587.35,Z 348.318,A -85,B 0,C 180,E1 -1281.046,E2 -1281.046} C_VEL
LIN {X 0,Y 587.33,Z 348.323,A -85,B 0,C 180,E1 -1284.007,E2 -1284.007} C_VEL
LIN {X 0,Y 587.356,Z 348.324,A -85,B 0,C 180,E1 -1286.278,E2 -1286.278} C_VEL
LIN {X 0,Y 587.344,Z 348.317,A -85,B 0,C 180,E1 -1289.135,E2 -1289.135} C_VEL
LIN {X 0,Y 587.352,Z 348.32,A -85,B 0,C 180,E1 -1291.839,E2 -1291.839} C_VEL
LIN {X 0,Y 587.348,Z 348.324,A -85,B 0,C 180,E1 -1294.35,E2 -1294.35} C_VEL
LIN {X 0,Y 587.349,Z 348.318,A -85,B 0,C 180,E1 -1296.747,E2 -1296.747} C_VEL
LIN {X 0,Y 587.343,Z 348.318,A -85,B 0,C 180,E1 -1299.36,E2 -1299.36} C_VEL
LIN {X 0,Y 587.331,Z 348.327,A -85,B 0,C 180,E1 -1302.109,E2 -1302.109} C_VEL
LIN {X 0,Y 587.313,Z 348.322,A -85,B 0,C 180,E1 -1304.912,E2 -1304.912} C_VEL
LIN {X 0,Y 587.352,Z 348.327,A -85,B 0,C 180,E1 -1307.929,E2 -1307.929} C_VEL
LIN {X 0,Y 587.335,Z 348.319,A -85,B 0,C 180,E1 -1311.059,E2 -1311.059} C_VEL
LIN {X 0,Y 587.355,Z 348.319,A -85,B 0,C 180,E1 -1313.293,E2 -1313.293} C_VEL
LIN {X 0,Y 587.37,Z 348.324,A -85,B 0,C 180,E1 -1315.781,E2 -1315.781} C_VEL
LIN {X 0,Y 587.345,Z 348.32,A -85,B 0,C 180,E1 -1318.232,E2 -1318.232} C_VEL
LIN {X 0,Y 587.355,Z 348.317,A -85,B 0,C 180,E1 -1320.867,E2 -1320.867} C_VEL
LIN {X 0,Y 587.371,Z 348.415,A -85,B 0,C 180,E1 -1322.789,E2 -1322.789} C_VEL
LIN {X 0,Y 587.398,Z 360.771,A -85,B 0,C 180,E1 -1325.055,E2 -1325.055} C_VEL
LIN {X 0,Y 587.331,Z 374.647,A -85,B 0,C 180,E1 -1327.568,E2 -1327.568} C_VEL
LIN {X 0,Y 587.864,Z 379.888,A -85,B 0,C 180,E1 -1327.647,E2 -1327.647} C_VEL
LIN {X 0,Y 587.722,Z 481.381,A -85,B 0,C 180,E1 -1328.908,E2 -1328.908} C_VEL
LIN {X 0,Y 587.656,Z 494.189,A -85,B 0,C 180,E1 -1329.204,E2 -1329.204} C_VEL
LIN {X 0,Y 587.625,Z 507.408,A -85,B 0,C 180,E1 -1329.661,E2 -1329.661} C_VEL
LIN {X 0,Y 587.526,Z 519.799,A -85,B 0,C 180,E1 -1330.25,E2 -1330.25} C_VEL
LIN {X 0,Y 587.428,Z 531.044,A -85,B 0,C 180,E1 -1330.938,E2 -1330.938} C_VEL
LIN {X 0,Y 587.392,Z 542.058,A -85,B 0,C 180,E1 -1331.786,E2 -1331.786} C_VEL
LIN {X 0,Y 587.28,Z 552.243,A -85,B 0,C 180,E1 -1332.77,E2 -1332.77} C_VEL
LIN {X 0,Y 587.251,Z 559.791,A -85,B 0,C 180,E1 -1333.666,E2 -1333.666} C_VEL
LIN {X 0,Y 587.219,Z 567.122,A -85,B 0,C 180,E1 -1334.734,E2 -1334.734} C_VEL
LIN {X 0,Y 587.196,Z 572.955,A -85,B 0,C 180,E1 -1335.807,E2 -1335.807} C_VEL
LIN {X 0,Y 587.166,Z 577.42,A -85,B 0,C 180,E1 -1336.855,E2 -1336.855} C_VEL
LIN {X 0,Y 587.181,Z 579.787,A -85,B 0,C 180,E1 -1337.559,E2 -1337.559} C_VEL
LIN {X 0,Y 587.162,Z 581.707,A -85,B 0,C 180,E1 -1338.26,E2 -1338.26} C_VEL
LIN {X 0,Y 587.169,Z 583.155,A -85,B 0,C 180,E1 -1338.959,E2 -1338.959} C_VEL
LIN {X 0,Y 587.151,Z 584.781,A -85,B 0,C 180,E1 -1340.353,E2 -1340.353} C_VEL
LIN {X 0,Y 587.127,Z 585,A -85,B 0,C 180,E1 -1341.048,E2 -1341.048} C_VEL
LIN {X 0,Y 587.146,Z 584.165,A -85,B 0,C 180,E1 -1342.434,E2 -1342.434} C_VEL
LIN {X 0,Y 587.189,Z 582.58,A -85,B 0,C 180,E1 -1343.427,E2 -1343.427} C_VEL
LIN {X 0,Y 587.157,Z 578.798,A -85,B 0,C 180,E1 -1344.85,E2 -1344.85} C_VEL
LIN {X 0,Y 587.183,Z 574.82,A -85,B 0,C 180,E1 -1345.882,E2 -1345.882} C_VEL
LIN {X 0,Y 587.236,Z 568.71,A -85,B 0,C 180,E1 -1347.085,E2 -1347.085} C_VEL
LIN {X 0,Y 587.253,Z 562.072,A -85,B 0,C 180,E1 -1348.114,E2 -1348.114} C_VEL
LIN {X 0,Y 587.307,Z 553.861,A -85,B 0,C 180,E1 -1349.143,E2 -1349.143} C_VEL
LIN {X 0,Y 587.33,Z 545.474,A -85,B 0,C 180,E1 -1350,E2 -1350} C_VEL
LIN {X 0,Y 587.399,Z 535.159,A -85,B 0,C 180,E1 -1350.857,E2 -1350.857} C_VEL
LIN {X 0,Y 587.457,Z 523.594,A -85,B 0,C 180,E1 -1351.628,E2 -1351.628} C_VEL
LIN {X 0,Y 587.562,Z 512.051,A -85,B 0,C 180,E1 -1352.228,E2 -1352.228} C_VEL
LIN {X 0,Y 587.606,Z 498.902,A -85,B 0,C 180,E1 -1352.742,E2 -1352.742} C_VEL
LIN {X 0,Y 587.672,Z 486.384,A -85,B 0,C 180,E1 -1353.085,E2 -1353.085} C_VEL
LIN {X 0,Y 587.73,Z 471.592,A -85,B 0,C 180,E1 -1353.32,E2 -1353.32} C_VEL
LIN {X 0,Y 587.815,Z 377.752,A -85,B 0,C 180,E1 -1354.471,E2 -1354.471} C_VEL
LIN {X 0,Y 587.323,Z 374.632,A -85,B 0,C 180,E1 -1354.525,E2 -1354.525} C_VEL
LIN {X 0,Y 587.409,Z 359.771,A -85,B 0,C 180,E1 -1357.217,E2 -1357.217} C_VEL
LIN {X 0,Y 587.358,Z 348.319,A -85,B 0,C 180,E1 -1359.339,E2 -1359.339} C_VEL
LIN {X 0,Y 587.341,Z 348.319,A -85,B 0,C 180,E1 -1361.737,E2 -1361.737} C_VEL
LIN {X 0,Y 587.345,Z 348.325,A -85,B 0,C 180,E1 -1364.553,E2 -1364.553} C_VEL
LIN {X 0,Y 587.355,Z 348.316,A -85,B 0,C 180,E1 -1367.405,E2 -1367.405} C_VEL
LIN {X 0,Y 587.335,Z 348.329,A -85,B 0,C 180,E1 -1370.304,E2 -1370.304} C_VEL
LIN {X 0,Y 587.327,Z 348.319,A -85,B 0,C 180,E1 -1373.258,E2 -1373.258} C_VEL
LIN {X 0,Y 587.337,Z 348.319,A -85,B 0,C 180,E1 -1375.516,E2 -1375.516} C_VEL
LIN {X 0,Y 587.352,Z 348.321,A -85,B 0,C 180,E1 -1377.817,E2 -1377.817} C_VEL
LIN {X 0,Y 587.348,Z 348.321,A -85,B 0,C 180,E1 -1380.511,E2 -1380.511} C_VEL
LIN {X 0,Y 587.336,Z 348.32,A -85,B 0,C 180,E1 -1383.396,E2 -1383.396} C_VEL
LIN {X 0,Y 587.358,Z 348.324,A -85,B 0,C 180,E1 -1385.894,E2 -1385.894} C_VEL
LIN {X 0,Y 587.333,Z 348.321,A -85,B 0,C 180,E1 -1388.478,E2 -1388.478} C_VEL
LIN {X 0,Y 587.334,Z 348.319,A -85,B 0,C 180,E1 -1391.156,E2 -1391.156} C_VEL
LIN {X 0,Y 587.324,Z 348.326,A -85,B 0,C 180,E1 -1394.112,E2 -1394.112} C_VEL
LIN {X 0,Y 587.32,Z 348.321,A -85,B 0,C 180,E1 -1396.994,E2 -1396.994} C_VEL
LIN {X 0,Y 587.315,Z 348.331,A -85,B 0,C 180,E1 -1399.745,E2 -1399.745} C_VEL
LIN {X 0,Y 587.342,Z 348.319,A -85,B 0,C 180,E1 -1402.392,E2 -1402.392} C_VEL
LIN {X 0,Y 587.322,Z 348.321,A -85,B 0,C 180,E1 -1404.944,E2 -1404.944} C_VEL
LIN {X 0,Y 587.338,Z 348.325,A -85,B 0,C 180,E1 -1407.42,E2 -1407.42} C_VEL
LIN {X 0,Y 587.328,Z 348.325,A -85,B 0,C 180,E1 -1409.829,E2 -1409.829} C_VEL
LIN {X 0,Y 587.345,Z 348.318,A -85,B 0,C 180,E1 -1412.306,E2 -1412.306} C_VEL
LIN {X 0,Y 587.331,Z 348.319,A -85,B 0,C 180,E1 -1414.483,E2 -1414.483} C_VEL
LIN {X 0,Y 587.362,Z 348.325,A -85,B 0,C 180,E1 -1417.487,E2 -1417.487} C_VEL
LIN {X 0,Y 587.339,Z 348.318,A -85,B 0,C 180,E1 -1420.425,E2 -1420.425} C_VEL
LIN {X 0,Y 587.351,Z 348.326,A -85,B 0,C 180,E1 -1423.311,E2 -1423.311} C_VEL
LIN {X 0,Y 587.353,Z 348.317,A -85,B 0,C 180,E1 -1426.154,E2 -1426.154} C_VEL
LIN {X 0,Y 587.343,Z 348.324,A -85,B 0,C 180,E1 -1428.962,E2 -1428.962} C_VEL
LIN {X 0,Y 587.365,Z 348.317,A -85,B 0,C 180,E1 -1431.744,E2 -1431.744} C_VEL
LIN {X 0,Y 587.357,Z 348.318,A -85,B 0,C 180,E1 -1434.507,E2 -1434.507} C_VEL
LIN {X 0,Y 587.378,Z 348.32,A -85,B 0,C 180,E1 -1437.257,E2 -1437.257} C_VEL
LIN {X 0,Y 587.373,Z 348.314,A -85,B 0,C 180,E1 -1440,E2 -1440} C_VEL
LIN {X 0,Y 587.378,Z 348.32,A -85,B 0,C 180,E1 -1442.743,E2 -1442.743} C_VEL
LIN {X 0,Y 587.357,Z 348.318,A -85,B 0,C 180,E1 -1445.493,E2 -1445.493} C_VEL
LIN {X 0,Y 587.364,Z 348.317,A -85,B 0,C 180,E1 -1448.255,E2 -1448.255} C_VEL
LIN {X 0,Y 587.352,Z 348.321,A -85,B 0,C 180,E1 -1451.141,E2 -1451.141} C_VEL
LIN {X 0,Y 587.355,Z 348.319,A -85,B 0,C 180,E1 -1454.261,E2 -1454.261} C_VEL
LIN {X 0,Y 587.354,Z 348.317,A -85,B 0,C 180,E1 -1457.406,E2 -1457.406} C_VEL
LIN {X 0,Y 587.33,Z 348.324,A -85,B 0,C 180,E1 -1460.305,E2 -1460.305} C_VEL
LIN {X 0,Y 587.359,Z 348.317,A -85,B 0,C 180,E1 -1463.257,E2 -1463.257} C_VEL
LIN {X 0,Y 587.355,Z 348.322,A -85,B 0,C 180,E1 -1466.278,E2 -1466.278} C_VEL
LIN {X 0,Y 587.345,Z 348.319,A -85,B 0,C 180,E1 -1469.135,E2 -1469.135} C_VEL
LIN {X 0,Y 587.352,Z 348.318,A -85,B 0,C 180,E1 -1471.839,E2 -1471.839} C_VEL
LIN {X 0,Y 587.348,Z 348.327,A -85,B 0,C 180,E1 -1474.35,E2 -1474.35} C_VEL
LIN {X 0,Y 587.347,Z 348.321,A -85,B 0,C 180,E1 -1476.747,E2 -1476.747} C_VEL
LIN {X 0,Y 587.339,Z 348.318,A -85,B 0,C 180,E1 -1479.36,E2 -1479.36} C_VEL
LIN {X 0,Y 587.329,Z 348.327,A -85,B 0,C 180,E1 -1482.108,E2 -1482.108} C_VEL
LIN {X 0,Y 587.311,Z 348.322,A -85,B 0,C 180,E1 -1484.912,E2 -1484.912} C_VEL
LIN {X 0,Y 587.349,Z 348.323,A -85,B 0,C 180,E1 -1487.928,E2 -1487.928} C_VEL
LIN {X 0,Y 587.332,Z 348.319,A -85,B 0,C 180,E1 -1491.059,E2 -1491.059} C_VEL
LIN {X 0,Y 587.352,Z 348.317,A -85,B 0,C 180,E1 -1493.292,E2 -1493.292} C_VEL
LIN {X 0,Y 587.368,Z 348.321,A -85,B 0,C 180,E1 -1495.781,E2 -1495.781} C_VEL
LIN {X 0,Y 587.352,Z 348.322,A -85,B 0,C 180,E1 -1498.233,E2 -1498.233} C_VEL
LIN {X 0,Y 587.351,Z 348.317,A -85,B 0,C 180,E1 -1500.867,E2 -1500.867} C_VEL
LIN {X 0,Y 587.361,Z 348.325,A -85,B 0,C 180,E1 -1503.819,E2 -1503.819} C_VEL
LIN {X 0,Y 587.387,Z 348.483,A -85,B 0,C 180,E1 -1506.418,E2 -1506.418} C_VEL
LIN {X 0,Y 587.915,Z 352.438,A -85,B 0,C 180,E1 -1506.995,E2 -1506.995} C_VEL
LIN {X 0,Y 587.737,Z 373.413,A -85,B 0,C 180,E1 -1509.893,E2 -1509.893} C_VEL
LIN {X 0,Y 587.601,Z 395.712,A -85,B 0,C 180,E1 -1512.92,E2 -1512.92} C_VEL
LIN {X 0,Y 587.478,Z 418.698,A -85,B 0,C 180,E1 -1515.991,E2 -1515.991} C_VEL
LIN {X 0,Y 587.407,Z 422.524,A -85,B 0,C 180,E1 -1516.497,E2 -1516.497} C_VEL
LIN {X 0,Y 587.899,Z 426.745,A -85,B 0,C 180,E1 -1516.564,E2 -1516.564} C_VEL
LIN {X 0,Y 587.744,Z 530.961,A -85,B 0,C 180,E1 -1517.856,E2 -1517.856} C_VEL
LIN {X 0,Y 587.668,Z 544.228,A -85,B 0,C 180,E1 -1518.161,E2 -1518.161} C_VEL
LIN {X 0,Y 587.616,Z 556.817,A -85,B 0,C 180,E1 -1518.592,E2 -1518.592} C_VEL
LIN {X 0,Y 587.552,Z 568.636,A -85,B 0,C 180,E1 -1519.141,E2 -1519.141} C_VEL
LIN {X 0,Y 587.465,Z 580.205,A -85,B 0,C 180,E1 -1519.837,E2 -1519.837} C_VEL
LIN {X 0,Y 587.391,Z 590.6,A -85,B 0,C 180,E1 -1520.618,E2 -1520.618} C_VEL
LIN {X 0,Y 587.321,Z 599.114,A -85,B 0,C 180,E1 -1521.398,E2 -1521.398} C_VEL
LIN {X 0,Y 587.273,Z 606.962,A -85,B 0,C 180,E1 -1522.263,E2 -1522.263} C_VEL
LIN {X 0,Y 587.23,Z 613.47,A -85,B 0,C 180,E1 -1523.126,E2 -1523.126} C_VEL
LIN {X 0,Y 587.236,Z 619.867,A -85,B 0,C 180,E1 -1524.161,E2 -1524.161} C_VEL
LIN {X 0,Y 587.147,Z 624.95,A -85,B 0,C 180,E1 -1525.194,E2 -1525.194} C_VEL
LIN {X 0,Y 587.212,Z 628.896,A -85,B 0,C 180,E1 -1526.226,E2 -1526.226} C_VEL
LIN {X 0,Y 587.132,Z 631.809,A -85,B 0,C 180,E1 -1527.256,E2 -1527.256} C_VEL
LIN {X 0,Y 587.139,Z 633.2,A -85,B 0,C 180,E1 -1527.942,E2 -1527.942} C_VEL
LIN {X 0,Y 587.14,Z 634.784,A -85,B 0,C 180,E1 -1529.314,E2 -1529.314} C_VEL
LIN {X 0,Y 587.137,Z 635,A -85,B 0,C 180,E1 -1530,E2 -1530} C_VEL
LIN {X 0,Y 587.147,Z 634.185,A -85,B 0,C 180,E1 -1531.372,E2 -1531.372} C_VEL
LIN {X 0,Y 587.139,Z 633.201,A -85,B 0,C 180,E1 -1532.058,E2 -1532.058} C_VEL
LIN {X 0,Y 587.132,Z 631.81,A -85,B 0,C 180,E1 -1532.744,E2 -1532.744} C_VEL
LIN {X 0,Y 587.212,Z 628.896,A -85,B 0,C 180,E1 -1533.774,E2 -1533.774} C_VEL
LIN {X 0,Y 587.147,Z 624.95,A -85,B 0,C 180,E1 -1534.806,E2 -1534.806} C_VEL
LIN {X 0,Y 587.217,Z 618.878,A -85,B 0,C 180,E1 -1536.011,E2 -1536.011} C_VEL
LIN {X 0,Y 587.245,Z 612.238,A -85,B 0,C 180,E1 -1537.046,E2 -1537.046} C_VEL
LIN {X 0,Y 587.299,Z 603.992,A -85,B 0,C 180,E1 -1538.083,E2 -1538.083} C_VEL
LIN {X 0,Y 587.343,Z 595.54,A -85,B 0,C 180,E1 -1538.949,E2 -1538.949} C_VEL
LIN {X 0,Y 587.416,Z 585.098,A -85,B 0,C 180,E1 -1539.816,E2 -1539.816} C_VEL
LIN {X 0,Y 587.496,Z 574.762,A -85,B 0,C 180,E1 -1540.511,E2 -1540.511} C_VEL
LIN {X 0,Y 587.583,Z 562.811,A -85,B 0,C 180,E1 -1541.149,E2 -1541.149} C_VEL
LIN {X 0,Y 587.624,Z 550.601,A -85,B 0,C 180,E1 -1541.639,E2 -1541.639} C_VEL
LIN {X 0,Y 587.696,Z 537.447,A -85,B 0,C 180,E1 -1542.014,E2 -1542.014} C_VEL
LIN {X 0,Y 587.774,Z 525.105,A -85,B 0,C 180,E1 -1542.231,E2 -1542.231} C_VEL
LIN {X 0,Y 587.731,Z 424.509,A -85,B 0,C 180,E1 -1543.467,E2 -1543.467} C_VEL
LIN {X 0,Y 587.409,Z 422.441,A -85,B 0,C 180,E1 -1543.513,E2 -1543.513} C_VEL
LIN {X 0,Y 587.554,Z 401.334,A -85,B 0,C 180,E1 -1546.325,E2 -1546.325} C_VEL
LIN {X 0,Y 587.736,Z 378.407,A -85,B 0,C 180,E1 -1549.424,E2 -1549.424} C_VEL
LIN {X 0,Y 587.899,Z 356.128,A -85,B 0,C 180,E1 -1552.491,E2 -1552.491} C_VEL
LIN {X 0,Y 587.824,Z 350.81,A -85,B 0,C 180,E1 -1553.237,E2 -1553.237} C_VEL
LIN {X 0,Y 587.347,Z 348.324,A -85,B 0,C 180,E1 -1553.631,E2 -1553.631} C_VEL
LIN {X 0,Y 587.34,Z 348.327,A -85,B 0,C 180,E1 -1556.278,E2 -1556.278} C_VEL
LIN {X 0,Y 587.351,Z 348.317,A -85,B 0,C 180,E1 -1559.133,E2 -1559.133} C_VEL
LIN {X 0,Y 587.354,Z 348.322,A -85,B 0,C 180,E1 -1561.837,E2 -1561.837} C_VEL
LIN {X 0,Y 587.357,Z 348.32,A -85,B 0,C 180,E1 -1564.349,E2 -1564.349} C_VEL
LIN {X 0,Y 587.351,Z 348.317,A -85,B 0,C 180,E1 -1566.746,E2 -1566.746} C_VEL
LIN {X 0,Y 587.344,Z 348.319,A -85,B 0,C 180,E1 -1569.358,E2 -1569.358} C_VEL
LIN {X 0,Y 587.331,Z 348.324,A -85,B 0,C 180,E1 -1572.107,E2 -1572.107} C_VEL
LIN {X 0,Y 587.311,Z 348.322,A -85,B 0,C 180,E1 -1575.088,E2 -1575.088} C_VEL
LIN {X 0,Y 587.347,Z 348.323,A -85,B 0,C 180,E1 -1577.927,E2 -1577.927} C_VEL
LIN {X 0,Y 587.329,Z 348.32,A -85,B 0,C 180,E1 -1581.057,E2 -1581.057} C_VEL
LIN {X 0,Y 587.348,Z 348.321,A -85,B 0,C 180,E1 -1583.291,E2 -1583.291} C_VEL
LIN {X 0,Y 587.361,Z 348.321,A -85,B 0,C 180,E1 -1585.78,E2 -1585.78} C_VEL
LIN {X 0,Y 587.35,Z 348.317,A -85,B 0,C 180,E1 -1588.232,E2 -1588.232} C_VEL
LIN {X 0,Y 587.347,Z 348.318,A -85,B 0,C 180,E1 -1590.865,E2 -1590.865} C_VEL
LIN {X 0,Y 587.354,Z 348.318,A -85,B 0,C 180,E1 -1593.818,E2 -1593.818} C_VEL
LIN {X 0,Y 587.359,Z 348.316,A -85,B 0,C 180,E1 -1596.743,E2 -1596.743} C_VEL
LIN {X 0,Y 587.33,Z 348.322,A -85,B 0,C 180,E1 -1599.695,E2 -1599.695} C_VEL
LIN {X 0,Y 587.354,Z 348.317,A -85,B 0,C 180,E1 -1602.594,E2 -1602.594} C_VEL
LIN {X 0,Y 587.355,Z 348.317,A -85,B 0,C 180,E1 -1605.739,E2 -1605.739} C_VEL
LIN {X 0,Y 587.352,Z 348.322,A -85,B 0,C 180,E1 -1608.859,E2 -1608.859} C_VEL
LIN {X 0,Y 587.364,Z 348.315,A -85,B 0,C 180,E1 -1611.745,E2 -1611.745} C_VEL
LIN {X 0,Y 587.358,Z 348.318,A -85,B 0,C 180,E1 -1614.507,E2 -1614.507} C_VEL
LIN {X 0,Y 587.377,Z 348.317,A -85,B 0,C 180,E1 -1617.257,E2 -1617.257} C_VEL
LIN {X 0,Y 587.373,Z 348.313,A -85,B 0,C 180,E1 -1620,E2 -1620} C_VEL
LIN {X 0,Y 587.378,Z 348.322,A -85,B 0,C 180,E1 -1622.743,E2 -1622.743} C_VEL
LIN {X 0,Y 587.355,Z 348.316,A -85,B 0,C 180,E1 -1625.493,E2 -1625.493} C_VEL
LIN {X 0,Y 587.365,Z 348.317,A -85,B 0,C 180,E1 -1628.256,E2 -1628.256} C_VEL
LIN {X 0,Y 587.353,Z 348.318,A -85,B 0,C 180,E1 -1631.142,E2 -1631.142} C_VEL
LIN {X 0,Y 587.356,Z 348.32,A -85,B 0,C 180,E1 -1634.261,E2 -1634.261} C_VEL
LIN {X 0,Y 587.352,Z 348.316,A -85,B 0,C 180,E1 -1637.406,E2 -1637.406} C_VEL
LIN {X 0,Y 587.319,Z 348.323,A -85,B 0,C 180,E1 -1638.331,E2 -1638.331} C_VEL
LIN {X 0,Y 586.666,Z 348.406,A -85,B 0,C 180,E1 -1638.903,E2 -1638.903} C_VEL
LIN {X 0,Y 583.835,Z 348.756,A -85,B 0,C 180,E1 -1639.831,E2 -1639.831} C_VEL
LIN {X 0,Y 581.426,Z 349.062,A -85,B 0,C 180,E1 -1640.578,E2 -1640.578} C_VEL
LIN {X 0,Y 580.374,Z 349.186,A -85,B 0,C 180,E1 -1641.154,E2 -1641.154} C_VEL
LIN {X 0,Y 580.28,Z 349.197,A -85,B 0,C 180,E1 -1641.35,E2 -1641.35} C_VEL
LIN {X 0,Y 580.293,Z 349.205,A -85,B 0,C 180,E1 -1644.317,E2 -1644.317} C_VEL
LIN {X 0,Y 580.3,Z 349.198,A -85,B 0,C 180,E1 -1646.623,E2 -1646.623} C_VEL
LIN {X 0,Y 580.296,Z 349.195,A -85,B 0,C 180,E1 -1649.311,E2 -1649.311} C_VEL
LIN {X 0,Y 580.299,Z 349.205,A -85,B 0,C 180,E1 -1652.201,E2 -1652.201} C_VEL
LIN {X 0,Y 580.294,Z 349.198,A -85,B 0,C 180,E1 -1654.696,E2 -1654.696} C_VEL
LIN {X 0,Y 580.297,Z 349.195,A -85,B 0,C 180,E1 -1657.269,E2 -1657.269} C_VEL
LIN {X 0,Y 580.303,Z 349.201,A -85,B 0,C 180,E1 -1660.273,E2 -1660.273} C_VEL
LIN {X 0,Y 580.28,Z 349.198,A -85,B 0,C 180,E1 -1662.707,E2 -1662.707} C_VEL
LIN {X 0,Y 580.272,Z 349.204,A -85,B 0,C 180,E1 -1665.61,E2 -1665.61} C_VEL
LIN {X 0,Y 580.314,Z 349.198,A -85,B 0,C 180,E1 -1668.235,E2 -1668.235} C_VEL
LIN {X 0,Y 580.291,Z 349.197,A -85,B 0,C 180,E1 -1670.967,E2 -1670.967} C_VEL
LIN {X 0,Y 580.298,Z 349.202,A -85,B 0,C 180,E1 -1673.6,E2 -1673.6} C_VEL
LIN {X 0,Y 580.321,Z 349.196,A -85,B 0,C 180,E1 -1676.146,E2 -1676.146} C_VEL
LIN {X 0,Y 580.281,Z 349.198,A -85,B 0,C 180,E1 -1678.616,E2 -1678.616} C_VEL
LIN {X 0,Y 580.298,Z 349.198,A -85,B 0,C 180,E1 -1681.025,E2 -1681.025} C_VEL
LIN {X 0,Y 580.339,Z 349.291,A -85,B 0,C 180,E1 -1682.724,E2 -1682.724} C_VEL
LIN {X 0,Y 580.402,Z 360.102,A -85,B 0,C 180,E1 -1684.734,E2 -1684.734} C_VEL
LIN {X 0,Y 580.291,Z 374.645,A -85,B 0,C 180,E1 -1687.401,E2 -1687.401} C_VEL
LIN {X 0,Y 580.982,Z 379.858,A -85,B 0,C 180,E1 -1687.485,E2 -1687.485} C_VEL
LIN {X 0,Y 580.803,Z 481.383,A -85,B 0,C 180,E1 -1688.762,E2 -1688.762} C_VEL
LIN {X 0,Y 580.73,Z 494.176,A -85,B 0,C 180,E1 -1689.061,E2 -1689.061} C_VEL
LIN {X 0,Y 580.63,Z 506.788,A -85,B 0,C 180,E1 -1689.497,E2 -1689.497} C_VEL
LIN {X 0,Y 580.536,Z 519.366,A -85,B 0,C 180,E1 -1690.094,E2 -1690.094} C_VEL
LIN {X 0,Y 580.427,Z 531.038,A -85,B 0,C 180,E1 -1690.814,E2 -1690.814} C_VEL
LIN {X 0,Y 580.332,Z 541.784,A -85,B 0,C 180,E1 -1691.648,E2 -1691.648} C_VEL
LIN {X 0,Y 580.276,Z 551.2,A -85,B 0,C 180,E1 -1692.557,E2 -1692.557} C_VEL
LIN {X 0,Y 580.186,Z 558.907,A -85,B 0,C 180,E1 -1693.462,E2 -1693.462} C_VEL
LIN {X 0,Y 580.155,Z 566.424,A -85,B 0,C 180,E1 -1694.544,E2 -1694.544} C_VEL
LIN {X 0,Y 580.114,Z 572.951,A -85,B 0,C 180,E1 -1695.742,E2 -1695.742} C_VEL
LIN {X 0,Y 580.095,Z 578.289,A -85,B 0,C 180,E1 -1697.048,E2 -1697.048} C_VEL
LIN {X 0,Y 580.063,Z 581.423,A -85,B 0,C 180,E1 -1698.114,E2 -1698.114} C_VEL
LIN {X 0,Y 580.075,Z 583.141,A -85,B 0,C 180,E1 -1698.926,E2 -1698.926} C_VEL
LIN {X 0,Y 580.057,Z 584.707,A -85,B 0,C 180,E1 -1700.234,E2 -1700.234} C_VEL
LIN {X 0,Y 580.026,Z 584.982,A -85,B 0,C 180,E1 -1700.937,E2 -1700.937} C_VEL
LIN {X 0,Y 580.061,Z 584.851,A -85,B 0,C 180,E1 -1701.64,E2 -1701.64} C_VEL
LIN {X 0,Y 580.062,Z 583.34,A -85,B 0,C 180,E1 -1703.041,E2 -1703.041} C_VEL
LIN {X 0,Y 580.068,Z 581.991,A -85,B 0,C 180,E1 -1703.74,E2 -1703.74} C_VEL
LIN {X 0,Y 580.073,Z 579.138,A -85,B 0,C 180,E1 -1704.787,E2 -1704.787} C_VEL
LIN {X 0,Y 580.106,Z 575.27,A -85,B 0,C 180,E1 -1705.832,E2 -1705.832} C_VEL
LIN {X 0,Y 580.122,Z 570.286,A -85,B 0,C 180,E1 -1706.875,E2 -1706.875} C_VEL
LIN {X 0,Y 580.141,Z 564.049,A -85,B 0,C 180,E1 -1707.917,E2 -1707.917} C_VEL
LIN {X 0,Y 580.231,Z 556.266,A -85,B 0,C 180,E1 -1708.959,E2 -1708.959} C_VEL
LIN {X 0,Y 580.275,Z 546.608,A -85,B 0,C 180,E1 -1710,E2 -1710} C_VEL
LIN {X 0,Y 580.374,Z 536.606,A -85,B 0,C 180,E1 -1710.867,E2 -1710.867} C_VEL
LIN {X 0,Y 580.447,Z 525.363,A -85,B 0,C 180,E1 -1711.648,E2 -1711.648} C_VEL
LIN {X 0,Y 580.555,Z 514.349,A -85,B 0,C 180,E1 -1712.255,E2 -1712.255} C_VEL
LIN {X 0,Y 580.646,Z 502.1,A -85,B 0,C 180,E1 -1712.775,E2 -1712.775} C_VEL
LIN {X 0,Y 580.715,Z 489.113,A -85,B 0,C 180,E1 -1713.165,E2 -1713.165} C_VEL
LIN {X 0,Y 580.792,Z 476.614,A -85,B 0,C 180,E1 -1713.404,E2 -1713.404} C_VEL
LIN {X 0,Y 580.866,Z 378.194,A -85,B 0,C 180,E1 -1714.629,E2 -1714.629} C_VEL
LIN {X 0,Y 580.311,Z 374.645,A -85,B 0,C 180,E1 -1714.689,E2 -1714.689} C_VEL
LIN {X 0,Y 580.399,Z 360.383,A -85,B 0,C 180,E1 -1717.304,E2 -1717.304} C_VEL
LIN {X 0,Y 580.294,Z 349.2,A -85,B 0,C 180,E1 -1719.388,E2 -1719.388} C_VEL
LIN {X 0,Y 580.31,Z 349.197,A -85,B 0,C 180,E1 -1721.881,E2 -1721.881} C_VEL
LIN {X 0,Y 580.293,Z 349.2,A -85,B 0,C 180,E1 -1724.734,E2 -1724.734} C_VEL
LIN {X 0,Y 580.299,Z 349.196,A -85,B 0,C 180,E1 -1727.624,E2 -1727.624} C_VEL
LIN {X 0,Y 580.293,Z 349.198,A -85,B 0,C 180,E1 -1729.822,E2 -1729.822} C_VEL
LIN {X 0,Y 580.277,Z 349.204,A -85,B 0,C 180,E1 -1732.052,E2 -1732.052} C_VEL
LIN {X 0,Y 580.31,Z 349.194,A -85,B 0,C 180,E1 -1735.079,E2 -1735.079} C_VEL
LIN {X 0,Y 580.305,Z 349.204,A -85,B 0,C 180,E1 -1738.185,E2 -1738.185} C_VEL
LIN {X 0,Y 580.293,Z 349.197,A -85,B 0,C 180,E1 -1740.695,E2 -1740.695} C_VEL
LIN {X 0,Y 580.305,Z 349.195,A -85,B 0,C 180,E1 -1743.316,E2 -1743.316} C_VEL
LIN {X 0,Y 580.327,Z 349.198,A -85,B 0,C 180,E1 -1745.767,E2 -1745.767} C_VEL
LIN {X 0,Y 580.289,Z 349.203,A -85,B 0,C 180,E1 -1748.145,E2 -1748.145} C_VEL
LIN {X 0,Y 580.297,Z 349.195,A -85,B 0,C 180,E1 -1750.842,E2 -1750.842} C_VEL
LIN {X 0,Y 580.276,Z 349.205,A -85,B 0,C 180,E1 -1753.657,E2 -1753.657} C_VEL
LIN {X 0,Y 580.284,Z 349.198,A -85,B 0,C 180,E1 -1756.607,E2 -1756.607} C_VEL
LIN {X 0,Y 580.297,Z 349.197,A -85,B 0,C 180,E1 -1759.156,E2 -1759.156} C_VEL
LIN {X 0,Y 580.287,Z 349.203,A -85,B 0,C 180,E1 -1761.926,E2 -1761.926} C_VEL
LIN {X 0,Y 580.281,Z 349.198,A -85,B 0,C 180,E1 -1764.454,E2 -1764.454} C_VEL
LIN {X 0,Y 580.288,Z 349.198,A -85,B 0,C 180,E1 -1766.975,E2 -1766.975} C_VEL
LIN {X 0,Y 580.296,Z 349.203,A -85,B 0,C 180,E1 -1769.425,E2 -1769.425} C_VEL
LIN {X 0,Y 580.314,Z 349.195,A -85,B 0,C 180,E1 -1772.136,E2 -1772.136} C_VEL
LIN {X 0,Y 580.301,Z 349.197,A -85,B 0,C 180,E1 -1774.92,E2 -1774.92} C_VEL
LIN {X 0,Y 580.322,Z 349.199,A -85,B 0,C 180,E1 -1777.198,E2 -1777.198} C_VEL
LIN {X 0,Y 580.302,Z 349.195,A -85,B 0,C 180,E1 -1780.177,E2 -1780.177} C_VEL
LIN {X 0,Y 580.322,Z 349.199,A -85,B 0,C 180,E1 -1783.103,E2 -1783.103} C_VEL
LIN {X 0,Y 580.318,Z 349.194,A -85,B 0,C 180,E1 -1785.983,E2 -1785.983} C_VEL
LIN {X 0,Y 580.322,Z 349.196,A -85,B 0,C 180,E1 -1788.827,E2 -1788.827} C_VEL
LIN {X 0,Y 580.328,Z 349.195,A -85,B 0,C 180,E1 -1791.644,E2 -1791.644} C_VEL
LIN {X 0,Y 580.322,Z 349.194,A -85,B 0,C 180,E1 -1794.44,E2 -1794.44} C_VEL
LIN {X 0,Y 580.343,Z 349.197,A -85,B 0,C 180,E1 -1797.223,E2 -1797.223} C_VEL
LIN {X 0,Y 580.343,Z 349.19,A -85,B 0,C 180,E1 -1800,E2 -1800} C_VEL
LIN {X 0,Y 580.343,Z 349.197,A -85,B 0,C 180,E1 -1802.776,E2 -1802.776} C_VEL
LIN {X 0,Y 580.322,Z 349.194,A -85,B 0,C 180,E1 -1805.56,E2 -1805.56} C_VEL
LIN {X 0,Y 580.328,Z 349.194,A -85,B 0,C 180,E1 -1808.356,E2 -1808.356} C_VEL
LIN {X 0,Y 580.323,Z 349.196,A -85,B 0,C 180,E1 -1811.208,E2 -1811.208} C_VEL
LIN {X 0,Y 580.318,Z 349.194,A -85,B 0,C 180,E1 -1814.017,E2 -1814.017} C_VEL
LIN {X 0,Y 580.309,Z 349.201,A -85,B 0,C 180,E1 -1816.916,E2 -1816.916} C_VEL
LIN {X 0,Y 580.301,Z 349.195,A -85,B 0,C 180,E1 -1819.822,E2 -1819.822} C_VEL
LIN {X 0,Y 580.321,Z 349.199,A -85,B 0,C 180,E1 -1822.801,E2 -1822.801} C_VEL
LIN {X 0,Y 580.3,Z 349.197,A -85,B 0,C 180,E1 -1825.08,E2 -1825.08} C_VEL
LIN {X 0,Y 580.313,Z 349.195,A -85,B 0,C 180,E1 -1827.864,E2 -1827.864} C_VEL
LIN {X 0,Y 580.285,Z 349.203,A -85,B 0,C 180,E1 -1830.697,E2 -1830.697} C_VEL
LIN {X 0,Y 580.299,Z 349.195,A -85,B 0,C 180,E1 -1833.318,E2 -1833.318} C_VEL
LIN {X 0,Y 580.319,Z 349.194,A -85,B 0,C 180,E1 -1835.768,E2 -1835.768} C_VEL
LIN {X 0,Y 580.283,Z 349.204,A -85,B 0,C 180,E1 -1838.147,E2 -1838.147} C_VEL
LIN {X 0,Y 580.295,Z 349.197,A -85,B 0,C 180,E1 -1840.844,E2 -1840.844} C_VEL
LIN {X 0,Y 580.284,Z 349.199,A -85,B 0,C 180,E1 -1843.658,E2 -1843.658} C_VEL
LIN {X 0,Y 580.272,Z 349.201,A -85,B 0,C 180,E1 -1846.61,E2 -1846.61} C_VEL
LIN {X 0,Y 580.297,Z 349.195,A -85,B 0,C 180,E1 -1849.158,E2 -1849.158} C_VEL
LIN {X 0,Y 580.289,Z 349.204,A -85,B 0,C 180,E1 -1851.927,E2 -1851.927} C_VEL
LIN {X 0,Y 580.307,Z 349.197,A -85,B 0,C 180,E1 -1854.458,E2 -1854.458} C_VEL
LIN {X 0,Y 580.29,Z 349.196,A -85,B 0,C 180,E1 -1856.976,E2 -1856.976} C_VEL
LIN {X 0,Y 580.31,Z 349.196,A -85,B 0,C 180,E1 -1859.427,E2 -1859.427} C_VEL
LIN {X 0,Y 580.32,Z 349.199,A -85,B 0,C 180,E1 -1862.138,E2 -1862.138} C_VEL
LIN {X 0,Y 580.323,Z 349.196,A -85,B 0,C 180,E1 -1865.27,E2 -1865.27} C_VEL
LIN {X 0,Y 580.312,Z 349.314,A -85,B 0,C 180,E1 -1866.231,E2 -1866.231} C_VEL
LIN {X 0,Y 581.032,Z 354.158,A -85,B 0,C 180,E1 -1866.95,E2 -1866.95} C_VEL
LIN {X 0,Y 580.837,Z 373.413,A -85,B 0,C 180,E1 -1869.644,E2 -1869.644} C_VEL
LIN {X 0,Y 580.615,Z 394.819,A -85,B 0,C 180,E1 -1872.586,E2 -1872.586} C_VEL
LIN {X 0,Y 580.467,Z 416.36,A -85,B 0,C 180,E1 -1875.504,E2 -1875.504} C_VEL
LIN {X 0,Y 580.415,Z 422.524,A -85,B 0,C 180,E1 -1876.332,E2 -1876.332} C_VEL
LIN {X 0,Y 580.983,Z 428.534,A -85,B 0,C 180,E1 -1876.423,E2 -1876.423} C_VEL
LIN {X 0,Y 580.815,Z 530.961,A -85,B 0,C 180,E1 -1877.709,E2 -1877.709} C_VEL
LIN {X 0,Y 580.726,Z 544.229,A -85,B 0,C 180,E1 -1878.017,E2 -1878.017} C_VEL
LIN {X 0,Y 580.664,Z 556.38,A -85,B 0,C 180,E1 -1878.437,E2 -1878.437} C_VEL
LIN {X 0,Y 580.574,Z 568.634,A -85,B 0,C 180,E1 -1879.009,E2 -1879.009} C_VEL
LIN {X 0,Y 580.444,Z 580.206,A -85,B 0,C 180,E1 -1879.712,E2 -1879.712} C_VEL
LIN {X 0,Y 580.341,Z 590.602,A -85,B 0,C 180,E1 -1880.503,E2 -1880.503} C_VEL
LIN {X 0,Y 580.271,Z 599.114,A -85,B 0,C 180,E1 -1881.292,E2 -1881.292} C_VEL
LIN {X 0,Y 580.221,Z 606.962,A -85,B 0,C 180,E1 -1882.168,E2 -1882.168} C_VEL
LIN {X 0,Y 580.153,Z 614.651,A -85,B 0,C 180,E1 -1883.222,E2 -1883.222} C_VEL
LIN {X 0,Y 580.139,Z 621.681,A -85,B 0,C 180,E1 -1884.439,E2 -1884.439} C_VEL
LIN {X 0,Y 580.108,Z 626.372,A -85,B 0,C 180,E1 -1885.484,E2 -1885.484} C_VEL
LIN {X 0,Y 580.123,Z 629.957,A -85,B 0,C 180,E1 -1886.527,E2 -1886.527} C_VEL
LIN {X 0,Y 580.043,Z 631.809,A -85,B 0,C 180,E1 -1887.222,E2 -1887.222} C_VEL
LIN {X 0,Y 580.038,Z 633.199,A -85,B 0,C 180,E1 -1887.917,E2 -1887.917} C_VEL
LIN {X 0,Y 580.04,Z 634.785,A -85,B 0,C 180,E1 -1889.306,E2 -1889.306} C_VEL
LIN {X 0,Y 580.037,Z 635,A -85,B 0,C 180,E1 -1890,E2 -1890} C_VEL
LIN {X 0,Y 580.047,Z 634.186,A -85,B 0,C 180,E1 -1891.389,E2 -1891.389} C_VEL
LIN {X 0,Y 580.038,Z 633.2,A -85,B 0,C 180,E1 -1892.083,E2 -1892.083} C_VEL
LIN {X 0,Y 580.043,Z 631.81,A -85,B 0,C 180,E1 -1892.778,E2 -1892.778} C_VEL
LIN {X 0,Y 580.109,Z 628.896,A -85,B 0,C 180,E1 -1893.82,E2 -1893.82} C_VEL
LIN {X 0,Y 580.054,Z 624.95,A -85,B 0,C 180,E1 -1894.865,E2 -1894.865} C_VEL
LIN {X 0,Y 580.139,Z 618.878,A -85,B 0,C 180,E1 -1896.085,E2 -1896.085} C_VEL
LIN {X 0,Y 580.184,Z 612.238,A -85,B 0,C 180,E1 -1897.132,E2 -1897.132} C_VEL
LIN {X 0,Y 580.25,Z 603.992,A -85,B 0,C 180,E1 -1898.182,E2 -1898.182} C_VEL
LIN {X 0,Y 580.308,Z 595.54,A -85,B 0,C 180,E1 -1899.058,E2 -1899.058} C_VEL
LIN {X 0,Y 580.417,Z 585.1,A -85,B 0,C 180,E1 -1899.936,E2 -1899.936} C_VEL
LIN {X 0,Y 580.507,Z 574.76,A -85,B 0,C 180,E1 -1900.639,E2 -1900.639} C_VEL
LIN {X 0,Y 580.596,Z 563.241,A -85,B 0,C 180,E1 -1901.264,E2 -1901.264} C_VEL
LIN {X 0,Y 580.664,Z 550.479,A -85,B 0,C 180,E1 -1901.785,E2 -1901.785} C_VEL
LIN {X 0,Y 580.743,Z 537.446,A -85,B 0,C 180,E1 -1902.16,E2 -1902.16} C_VEL
LIN {X 0,Y 580.859,Z 525.105,A -85,B 0,C 180,E1 -1902.379,E2 -1902.379} C_VEL
LIN {X 0,Y 580.815,Z 425.182,A -85,B 0,C 180,E1 -1903.622,E2 -1903.622} C_VEL
LIN {X 0,Y 580.419,Z 422.441,A -85,B 0,C 180,E1 -1903.679,E2 -1903.679} C_VEL
LIN {X 0,Y 580.571,Z 400.004,A -85,B 0,C 180,E1 -1906.708,E2 -1906.708} C_VEL
LIN {X 0,Y 580.793,Z 377.402,A -85,B 0,C 180,E1 -1909.804,E2 -1909.804} C_VEL
LIN {X 0,Y 581.038,Z 356.128,A -85,B 0,C 180,E1 -1912.771,E2 -1912.771} C_VEL
LIN {X 0,Y 580.952,Z 352.486,A -85,B 0,C 180,E1 -1913.29,E2 -1913.29} C_VEL
LIN {X 0,Y 580.302,Z 349.202,A -85,B 0,C 180,E1 -1913.793,E2 -1913.793} C_VEL
LIN {X 0,Y 580.278,Z 349.201,A -85,B 0,C 180,E1 -1916.623,E2 -1916.623} C_VEL
LIN {X 0,Y 580.306,Z 349.195,A -85,B 0,C 180,E1 -1919.31,E2 -1919.31} C_VEL
LIN {X 0,Y 580.302,Z 349.202,A -85,B 0,C 180,E1 -1922.199,E2 -1922.199} C_VEL
LIN {X 0,Y 580.301,Z 349.196,A -85,B 0,C 180,E1 -1924.695,E2 -1924.695} C_VEL
LIN {X 0,Y 580.298,Z 349.196,A -85,B 0,C 180,E1 -1927.267,E2 -1927.267} C_VEL
LIN {X 0,Y 580.295,Z 349.199,A -85,B 0,C 180,E1 -1930.271,E2 -1930.271} C_VEL
LIN {X 0,Y 580.273,Z 349.198,A -85,B 0,C 180,E1 -1932.706,E2 -1932.706} C_VEL
LIN {X 0,Y 580.269,Z 349.206,A -85,B 0,C 180,E1 -1935.608,E2 -1935.608} C_VEL
LIN {X 0,Y 580.309,Z 349.195,A -85,B 0,C 180,E1 -1938.234,E2 -1938.234} C_VEL
LIN {X 0,Y 580.284,Z 349.197,A -85,B 0,C 180,E1 -1940.965,E2 -1940.965} C_VEL
LIN {X 0,Y 580.291,Z 349.206,A -85,B 0,C 180,E1 -1943.598,E2 -1943.598} C_VEL
LIN {X 0,Y 580.314,Z 349.195,A -85,B 0,C 180,E1 -1946.145,E2 -1946.145} C_VEL
LIN {X 0,Y 580.285,Z 349.197,A -85,B 0,C 180,E1 -1948.615,E2 -1948.615} C_VEL
LIN {X 0,Y 580.291,Z 349.199,A -85,B 0,C 180,E1 -1951.024,E2 -1951.024} C_VEL
LIN {X 0,Y 580.32,Z 349.196,A -85,B 0,C 180,E1 -1953.658,E2 -1953.658} C_VEL
LIN {X 0,Y 580.295,Z 349.194,A -85,B 0,C 180,E1 -1956.443,E2 -1956.443} C_VEL
LIN {X 0,Y 580.278,Z 349.204,A -85,B 0,C 180,E1 -1959.437,E2 -1959.437} C_VEL
LIN {X 0,Y 580.277,Z 349.201,A -85,B 0,C 180,E1 -1961.645,E2 -1961.645} C_VEL
LIN {X 0,Y 580.278,Z 349.198,A -85,B 0,C 180,E1 -1963.826,E2 -1963.826} C_VEL
LIN {X 0,Y 580.275,Z 349.201,A -85,B 0,C 180,E1 -1966.696,E2 -1966.696} C_VEL
LIN {X 0,Y 580.3,Z 349.197,A -85,B 0,C 180,E1 -1969.533,E2 -1969.533} C_VEL
LIN {X 0,Y 580.333,Z 349.192,A -85,B 0,C 180,E1 -1972.345,E2 -1972.345} C_VEL
LIN {X 0,Y 580.336,Z 349.197,A -85,B 0,C 180,E1 -1975.137,E2 -1975.137} C_VEL
LIN {X 0,Y 580.33,Z 349.191,A -85,B 0,C 180,E1 -1977.918,E2 -1977.918} C_VEL
LIN {X 0,Y 580.365,Z 349.194,A -85,B 0,C 180,E1 -1980.694,E2 -1980.694} C_VEL
LIN {X 0,Y 580.286,Z 349.197,A -85,B 0,C 180,E1 -1983.472,E2 -1983.472} C_VEL
LIN {X 0,Y 580.32,Z 349.193,A -85,B 0,C 180,E1 -1985.56,E2 -1985.56} C_VEL
LIN {X 0,Y 580.328,Z 349.195,A -85,B 0,C 180,E1 -1988.356,E2 -1988.356} C_VEL
LIN {X 0,Y 580.324,Z 349.193,A -85,B 0,C 180,E1 -1991.209,E2 -1991.209} C_VEL
LIN {X 0,Y 580.318,Z 349.194,A -85,B 0,C 180,E1 -1994.017,E2 -1994.017} C_VEL
LIN {X 0,Y 580.306,Z 349.197,A -85,B 0,C 180,E1 -1996.916,E2 -1996.916} C_VEL
LIN {X 0,Y 580.3,Z 349.196,A -85,B 0,C 180,E1 -1999.823,E2 -1999.823} C_VEL
LIN {X 0,Y 580.28,Z 349.197,A -85,B 0,C 180,E1 -2001.35,E2 -2001.35} C_VEL
LIN {X 0,Y 579.583,Z 349.288,A -85,B 0,C 180,E1 -2001.929,E2 -2001.929} C_VEL
LIN {X 0,Y 576.705,Z 349.646,A -85,B 0,C 180,E1 -2002.868,E2 -2002.868} C_VEL
LIN {X 0,Y 574.309,Z 349.943,A -85,B 0,C 180,E1 -2003.625,E2 -2003.625} C_VEL
LIN {X 0,Y 573.31,Z 350.073,A -85,B 0,C 180,E1 -2004.209,E2 -2004.209} C_VEL
LIN {X 0,Y 573.244,Z 350.076,A -85,B 0,C 180,E1 -2004.406,E2 -2004.406} C_VEL
LIN {X 0,Y 573.258,Z 350.071,A -85,B 0,C 180,E1 -2006.976,E2 -2006.976} C_VEL
LIN {X 0,Y 573.242,Z 350.075,A -85,B 0,C 180,E1 -2009.489,E2 -2009.489} C_VEL
LIN {X 0,Y 573.252,Z 350.083,A -85,B 0,C 180,E1 -2012.23,E2 -2012.23} C_VEL
LIN {X 0,Y 573.245,Z 350.075,A -85,B 0,C 180,E1 -2014.775,E2 -2014.775} C_VEL
LIN {X 0,Y 573.25,Z 350.073,A -85,B 0,C 180,E1 -2017.167,E2 -2017.167} C_VEL
LIN {X 0,Y 573.246,Z 350.077,A -85,B 0,C 180,E1 -2019.608,E2 -2019.608} C_VEL
LIN {X 0,Y 573.241,Z 350.075,A -85,B 0,C 180,E1 -2022.643,E2 -2022.643} C_VEL
LIN {X 0,Y 573.237,Z 350.081,A -85,B 0,C 180,E1 -2025.668,E2 -2025.668} C_VEL
LIN {X 0,Y 573.245,Z 350.076,A -85,B 0,C 180,E1 -2028.545,E2 -2028.545} C_VEL
LIN {X 0,Y 573.25,Z 350.076,A -85,B 0,C 180,E1 -2031.3,E2 -2031.3} C_VEL
LIN {X 0,Y 573.266,Z 350.078,A -85,B 0,C 180,E1 -2034.012,E2 -2034.012} C_VEL
LIN {X 0,Y 573.287,Z 350.069,A -85,B 0,C 180,E1 -2036.52,E2 -2036.52} C_VEL
LIN {X 0,Y 573.237,Z 350.078,A -85,B 0,C 180,E1 -2039.118,E2 -2039.118} C_VEL
LIN {X 0,Y 573.243,Z 350.082,A -85,B 0,C 180,E1 -2041.437,E2 -2041.437} C_VEL
LIN {X 0,Y 573.304,Z 350.172,A -85,B 0,C 180,E1 -2042.657,E2 -2042.657} C_VEL
LIN {X 0,Y 573.365,Z 360.465,A -85,B 0,C 180,E1 -2044.596,E2 -2044.596} C_VEL
LIN {X 0,Y 573.257,Z 374.645,A -85,B 0,C 180,E1 -2047.23,E2 -2047.23} C_VEL
LIN {X 0,Y 574.077,Z 379.79,A -85,B 0,C 180,E1 -2047.318,E2 -2047.318} C_VEL
LIN {X 0,Y 573.863,Z 481.397,A -85,B 0,C 180,E1 -2048.611,E2 -2048.611} C_VEL
LIN {X 0,Y 573.769,Z 494.162,A -85,B 0,C 180,E1 -2048.913,E2 -2048.913} C_VEL
LIN {X 0,Y 573.659,Z 507.35,A -85,B 0,C 180,E1 -2049.377,E2 -2049.377} C_VEL
LIN {X 0,Y 573.573,Z 518.94,A -85,B 0,C 180,E1 -2049.936,E2 -2049.936} C_VEL
LIN {X 0,Y 573.42,Z 531.067,A -85,B 0,C 180,E1 -2050.69,E2 -2050.69} C_VEL
LIN {X 0,Y 573.312,Z 541.511,A -85,B 0,C 180,E1 -2051.507,E2 -2051.507} C_VEL
LIN {X 0,Y 573.233,Z 550.135,A -85,B 0,C 180,E1 -2052.336,E2 -2052.336} C_VEL
LIN {X 0,Y 573.146,Z 558.44,A -85,B 0,C 180,E1 -2053.307,E2 -2053.307} C_VEL
LIN {X 0,Y 573.049,Z 565.695,A -85,B 0,C 180,E1 -2054.347,E2 -2054.347} C_VEL
LIN {X 0,Y 573.028,Z 571.746,A -85,B 0,C 180,E1 -2055.427,E2 -2055.427} C_VEL
LIN {X 0,Y 573.017,Z 576.582,A -85,B 0,C 180,E1 -2056.525,E2 -2056.525} C_VEL
LIN {X 0,Y 572.991,Z 580.189,A -85,B 0,C 180,E1 -2057.606,E2 -2057.606} C_VEL
LIN {X 0,Y 572.987,Z 583.122,A -85,B 0,C 180,E1 -2058.888,E2 -2058.888} C_VEL
LIN {X 0,Y 572.974,Z 584.631,A -85,B 0,C 180,E1 -2060.112,E2 -2060.112} C_VEL
LIN {X 0,Y 572.951,Z 584.896,A -85,B 0,C 180,E1 -2061.536,E2 -2061.536} C_VEL
LIN {X 0,Y 572.978,Z 584.413,A -85,B 0,C 180,E1 -2062.246,E2 -2062.246} C_VEL
LIN {X 0,Y 573.013,Z 582.652,A -85,B 0,C 180,E1 -2063.451,E2 -2063.451} C_VEL
LIN {X 0,Y 572.993,Z 579.473,A -85,B 0,C 180,E1 -2064.722,E2 -2064.722} C_VEL
LIN {X 0,Y 573.032,Z 575.717,A -85,B 0,C 180,E1 -2065.78,E2 -2065.78} C_VEL
LIN {X 0,Y 573.035,Z 570.857,A -85,B 0,C 180,E1 -2066.836,E2 -2066.836} C_VEL
LIN {X 0,Y 573.056,Z 564.754,A -85,B 0,C 180,E1 -2067.892,E2 -2067.892} C_VEL
LIN {X 0,Y 573.172,Z 557.183,A -85,B 0,C 180,E1 -2068.946,E2 -2068.946} C_VEL
LIN {X 0,Y 573.222,Z 547.721,A -85,B 0,C 180,E1 -2070,E2 -2070} C_VEL
LIN {X 0,Y 573.35,Z 537.984,A -85,B 0,C 180,E1 -2070.878,E2 -2070.878} C_VEL
LIN {X 0,Y 573.433,Z 527.121,A -85,B 0,C 180,E1 -2071.668,E2 -2071.668} C_VEL
LIN {X 0,Y 573.571,Z 514.801,A -85,B 0,C 180,E1 -2072.37,E2 -2072.37} C_VEL
LIN {X 0,Y 573.674,Z 502.723,A -85,B 0,C 180,E1 -2072.897,E2 -2072.897} C_VEL
LIN {X 0,Y 573.772,Z 490.038,A -85,B 0,C 180,E1 -2073.291,E2 -2073.291} C_VEL
LIN {X 0,Y 573.877,Z 476.642,A -85,B 0,C 180,E1 -2073.554,E2 -2073.554} C_VEL
LIN {X 0,Y 573.963,Z 379.018,A -85,B 0,C 180,E1 -2074.785,E2 -2074.785} C_VEL
LIN {X 0,Y 573.318,Z 374.538,A -85,B 0,C 180,E1 -2074.878,E2 -2074.878} C_VEL
LIN {X 0,Y 573.386,Z 357.214,A -85,B 0,C 180,E1 -2078.103,E2 -2078.103} C_VEL
LIN {X 0,Y 573.269,Z 350.076,A -85,B 0,C 180,E1 -2079.459,E2 -2079.459} C_VEL
LIN {X 0,Y 573.279,Z 350.075,A -85,B 0,C 180,E1 -2082.029,E2 -2082.029} C_VEL
LIN {X 0,Y 573.241,Z 350.076,A -85,B 0,C 180,E1 -2084.919,E2 -2084.919} C_VEL
LIN {X 0,Y 573.25,Z 350.076,A -85,B 0,C 180,E1 -2087.848,E2 -2087.848} C_VEL
LIN {X 0,Y 573.248,Z 350.08,A -85,B 0,C 180,E1 -2090.076,E2 -2090.076} C_VEL
LIN {X 0,Y 573.241,Z 350.083,A -85,B 0,C 180,E1 -2092.337,E2 -2092.337} C_VEL
LIN {X 0,Y 573.258,Z 350.073,A -85,B 0,C 180,E1 -2095.409,E2 -2095.409} C_VEL
LIN {X 0,Y 573.267,Z 350.079,A -85,B 0,C 180,E1 -2098.031,E2 -2098.031} C_VEL
LIN {X 0,Y 573.237,Z 350.075,A -85,B 0,C 180,E1 -2100.882,E2 -2100.882} C_VEL
LIN {X 0,Y 573.263,Z 350.074,A -85,B 0,C 180,E1 -2103.523,E2 -2103.523} C_VEL
LIN {X 0,Y 573.262,Z 350.081,A -85,B 0,C 180,E1 -2106.047,E2 -2106.047} C_VEL
LIN {X 0,Y 573.249,Z 350.074,A -85,B 0,C 180,E1 -2108.7,E2 -2108.7} C_VEL
LIN {X 0,Y 573.228,Z 350.079,A -85,B 0,C 180,E1 -2111.456,E2 -2111.456} C_VEL
LIN {X 0,Y 573.233,Z 350.078,A -85,B 0,C 180,E1 -2114.332,E2 -2114.332} C_VEL
LIN {X 0,Y 573.241,Z 350.078,A -85,B 0,C 180,E1 -2117.357,E2 -2117.357} C_VEL
LIN {X 0,Y 573.243,Z 350.076,A -85,B 0,C 180,E1 -2120.392,E2 -2120.392} C_VEL
LIN {X 0,Y 573.251,Z 350.075,A -85,B 0,C 180,E1 -2123.077,E2 -2123.077} C_VEL
LIN {X 0,Y 573.263,Z 350.081,A -85,B 0,C 180,E1 -2125.671,E2 -2125.671} C_VEL
LIN {X 0,Y 573.245,Z 350.076,A -85,B 0,C 180,E1 -2128.184,E2 -2128.184} C_VEL
LIN {X 0,Y 573.26,Z 350.072,A -85,B 0,C 180,E1 -2130.633,E2 -2130.633} C_VEL
LIN {X 0,Y 573.263,Z 350.081,A -85,B 0,C 180,E1 -2133.5,E2 -2133.5} C_VEL
LIN {X 0,Y 573.237,Z 350.076,A -85,B 0,C 180,E1 -2136.134,E2 -2136.134} C_VEL
LIN {X 0,Y 573.253,Z 350.074,A -85,B 0,C 180,E1 -2138.706,E2 -2138.706} C_VEL
LIN {X 0,Y 573.233,Z 350.084,A -85,B 0,C 180,E1 -2141.411,E2 -2141.411} C_VEL
LIN {X 0,Y 573.253,Z 350.078,A -85,B 0,C 180,E1 -2143.622,E2 -2143.622} C_VEL
LIN {X 0,Y 573.232,Z 350.077,A -85,B 0,C 180,E1 -2146.529,E2 -2146.529} C_VEL
LIN {X 0,Y 573.269,Z 350.078,A -85,B 0,C 180,E1 -2149.403,E2 -2149.403} C_VEL
LIN {X 0,Y 573.282,Z 350.07,A -85,B 0,C 180,E1 -2152.25,E2 -2152.25} C_VEL
LIN {X 0,Y 573.308,Z 350.075,A -85,B 0,C 180,E1 -2155.077,E2 -2155.077} C_VEL
LIN {X 0,Y 573.301,Z 350.068,A -85,B 0,C 180,E1 -2157.892,E2 -2157.892} C_VEL
LIN {X 0,Y 573.333,Z 350.068,A -85,B 0,C 180,E1 -2160.702,E2 -2160.702} C_VEL
LIN {X 0,Y 573.237,Z 350.077,A -85,B 0,C 180,E1 -2163.514,E2 -2163.514} C_VEL
LIN {X 0,Y 573.288,Z 350.07,A -85,B 0,C 180,E1 -2165.628,E2 -2165.628} C_VEL
LIN {X 0,Y 573.3,Z 350.071,A -85,B 0,C 180,E1 -2168.459,E2 -2168.459} C_VEL
LIN {X 0,Y 573.289,Z 350.071,A -85,B 0,C 180,E1 -2171.312,E2 -2171.312} C_VEL
LIN {X 0,Y 573.271,Z 350.076,A -85,B 0,C 180,E1 -2174.425,E2 -2174.425} C_VEL
LIN {X 0,Y 573.253,Z 350.077,A -85,B 0,C 180,E1 -2177.112,E2 -2177.112} C_VEL
LIN {X 0,Y 573.25,Z 350.075,A -85,B 0,C 180,E1 -2180.077,E2 -2180.077} C_VEL
LIN {X 0,Y 573.263,Z 350.074,A -85,B 0,C 180,E1 -2183.154,E2 -2183.154} C_VEL
LIN {X 0,Y 573.281,Z 350.074,A -85,B 0,C 180,E1 -2186.189,E2 -2186.189} C_VEL
LIN {X 0,Y 573.236,Z 350.083,A -85,B 0,C 180,E1 -2188.565,E2 -2188.565} C_VEL
LIN {X 0,Y 573.23,Z 350.078,A -85,B 0,C 180,E1 -2190.993,E2 -2190.993} C_VEL
LIN {X 0,Y 573.281,Z 350.07,A -85,B 0,C 180,E1 -2193.529,E2 -2193.529} C_VEL
LIN {X 0,Y 573.254,Z 350.078,A -85,B 0,C 180,E1 -2196.049,E2 -2196.049} C_VEL
LIN {X 0,Y 573.243,Z 350.078,A -85,B 0,C 180,E1 -2198.702,E2 -2198.702} C_VEL
LIN {X 0,Y 573.248,Z 350.075,A -85,B 0,C 180,E1 -2201.596,E2 -2201.596} C_VEL
LIN {X 0,Y 573.235,Z 350.083,A -85,B 0,C 180,E1 -2204.334,E2 -2204.334} C_VEL
LIN {X 0,Y 573.236,Z 350.075,A -85,B 0,C 180,E1 -2207.359,E2 -2207.359} C_VEL
LIN {X 0,Y 573.246,Z 350.079,A -85,B 0,C 180,E1 -2210.394,E2 -2210.394} C_VEL
LIN {X 0,Y 573.254,Z 350.073,A -85,B 0,C 180,E1 -2213.079,E2 -2213.079} C_VEL
LIN {X 0,Y 573.274,Z 350.075,A -85,B 0,C 180,E1 -2215.673,E2 -2215.673} C_VEL
LIN {X 0,Y 573.249,Z 350.079,A -85,B 0,C 180,E1 -2218.186,E2 -2218.186} C_VEL
LIN {X 0,Y 573.269,Z 350.072,A -85,B 0,C 180,E1 -2220.635,E2 -2220.635} C_VEL
LIN {X 0,Y 573.252,Z 350.074,A -85,B 0,C 180,E1 -2223.025,E2 -2223.025} C_VEL
LIN {X 0,Y 573.267,Z 350.118,A -85,B 0,C 180,E1 -2226.065,E2 -2226.065} C_VEL
LIN {X 0,Y 574.068,Z 354.129,A -85,B 0,C 180,E1 -2226.662,E2 -2226.662} C_VEL
LIN {X 0,Y 573.941,Z 370.903,A -85,B 0,C 180,E1 -2229.034,E2 -2229.034} C_VEL
LIN {X 0,Y 573.677,Z 390.697,A -85,B 0,C 180,E1 -2231.797,E2 -2231.797} C_VEL
LIN {X 0,Y 573.494,Z 409.311,A -85,B 0,C 180,E1 -2234.36,E2 -2234.36} C_VEL
LIN {X 0,Y 573.412,Z 422.524,A -85,B 0,C 180,E1 -2236.161,E2 -2236.161} C_VEL
LIN {X 0,Y 574.089,Z 428.534,A -85,B 0,C 180,E1 -2236.257,E2 -2236.257} C_VEL
LIN {X 0,Y 573.879,Z 530.961,A -85,B 0,C 180,E1 -2237.558,E2 -2237.558} C_VEL
LIN {X 0,Y 573.799,Z 544.229,A -85,B 0,C 180,E1 -2237.87,E2 -2237.87} C_VEL
LIN {X 0,Y 573.713,Z 556.381,A -85,B 0,C 180,E1 -2238.295,E2 -2238.295} C_VEL
LIN {X 0,Y 573.574,Z 567.595,A -85,B 0,C 180,E1 -2238.817,E2 -2238.817} C_VEL
LIN {X 0,Y 573.469,Z 578.914,A -85,B 0,C 180,E1 -2239.497,E2 -2239.497} C_VEL
LIN {X 0,Y 573.345,Z 589.544,A -85,B 0,C 180,E1 -2240.297,E2 -2240.297} C_VEL
LIN {X 0,Y 573.241,Z 599.115,A -85,B 0,C 180,E1 -2241.185,E2 -2241.185} C_VEL
LIN {X 0,Y 573.161,Z 606.962,A -85,B 0,C 180,E1 -2242.071,E2 -2242.071} C_VEL
LIN {X 0,Y 573.072,Z 614.955,A -85,B 0,C 180,E1 -2243.185,E2 -2243.185} C_VEL
LIN {X 0,Y 573.07,Z 621.681,A -85,B 0,C 180,E1 -2244.37,E2 -2244.37} C_VEL
LIN {X 0,Y 573.029,Z 626.372,A -85,B 0,C 180,E1 -2245.428,E2 -2245.428} C_VEL
LIN {X 0,Y 573.022,Z 629.957,A -85,B 0,C 180,E1 -2246.484,E2 -2246.484} C_VEL
LIN {X 0,Y 572.959,Z 631.808,A -85,B 0,C 180,E1 -2247.188,E2 -2247.188} C_VEL
LIN {X 0,Y 572.938,Z 633.198,A -85,B 0,C 180,E1 -2247.891,E2 -2247.891} C_VEL
LIN {X 0,Y 572.941,Z 634.785,A -85,B 0,C 180,E1 -2249.297,E2 -2249.297} C_VEL
LIN {X 0,Y 572.938,Z 635,A -85,B 0,C 180,E1 -2250,E2 -2250} C_VEL
LIN {X 0,Y 572.946,Z 634.186,A -85,B 0,C 180,E1 -2251.406,E2 -2251.406} C_VEL
LIN {X 0,Y 572.938,Z 633.2,A -85,B 0,C 180,E1 -2252.109,E2 -2252.109} C_VEL
LIN {X 0,Y 572.959,Z 631.81,A -85,B 0,C 180,E1 -2252.812,E2 -2252.812} C_VEL
LIN {X 0,Y 573.014,Z 628.896,A -85,B 0,C 180,E1 -2253.868,E2 -2253.868} C_VEL
LIN {X 0,Y 572.963,Z 624.949,A -85,B 0,C 180,E1 -2254.925,E2 -2254.925} C_VEL
LIN {X 0,Y 573.064,Z 618.878,A -85,B 0,C 180,E1 -2256.16,E2 -2256.16} C_VEL
LIN {X 0,Y 573.119,Z 612.239,A -85,B 0,C 180,E1 -2257.221,E2 -2257.221} C_VEL
LIN {X 0,Y 573.201,Z 603.992,A -85,B 0,C 180,E1 -2258.283,E2 -2258.283} C_VEL
LIN {X 0,Y 573.286,Z 595.541,A -85,B 0,C 180,E1 -2259.17,E2 -2259.17} C_VEL
LIN {X 0,Y 573.423,Z 585.101,A -85,B 0,C 180,E1 -2260.058,E2 -2260.058} C_VEL
LIN {X 0,Y 573.528,Z 573.358,A -85,B 0,C 180,E1 -2260.858,E2 -2260.858} C_VEL
LIN {X 0,Y 573.652,Z 562.288,A -85,B 0,C 180,E1 -2261.447,E2 -2261.447} C_VEL
LIN {X 0,Y 573.745,Z 549.18,A -85,B 0,C 180,E1 -2261.974,E2 -2261.974} C_VEL
LIN {X 0,Y 573.841,Z 536.531,A -85,B 0,C 180,E1 -2262.331,E2 -2262.331} C_VEL
LIN {X 0,Y 573.922,Z 523.333,A -85,B 0,C 180,E1 -2262.554,E2 -2262.554} C_VEL
LIN {X 0,Y 573.984,Z 426.422,A -85,B 0,C 180,E1 -2263.772,E2 -2263.772} C_VEL
LIN {X 0,Y 573.418,Z 422.441,A -85,B 0,C 180,E1 -2263.85,E2 -2263.85} C_VEL
LIN {X 0,Y 573.622,Z 399.373,A -85,B 0,C 180,E1 -2267.004,E2 -2267.004} C_VEL
LIN {X 0,Y 573.869,Z 377.402,A -85,B 0,C 180,E1 -2270.054,E2 -2270.054} C_VEL
LIN {X 0,Y 574.13,Z 356.07,A -85,B 0,C 180,E1 -2273.061,E2 -2273.061} C_VEL
LIN {X 0,Y 573.576,Z 351.687,A -85,B 0,C 180,E1 -2273.697,E2 -2273.697} C_VEL
LIN {X 0,Y 573.265,Z 350.08,A -85,B 0,C 180,E1 -2273.959,E2 -2273.959} C_VEL
LIN {X 0,Y 573.252,Z 350.074,A -85,B 0,C 180,E1 -2276.975,E2 -2276.975} C_VEL
LIN {X 0,Y 573.253,Z 350.075,A -85,B 0,C 180,E1 -2279.489,E2 -2279.489} C_VEL
LIN {X 0,Y 573.255,Z 350.079,A -85,B 0,C 180,E1 -2282.228,E2 -2282.228} C_VEL
LIN {X 0,Y 573.252,Z 350.074,A -85,B 0,C 180,E1 -2284.773,E2 -2284.773} C_VEL
LIN {X 0,Y 573.252,Z 350.074,A -85,B 0,C 180,E1 -2287.165,E2 -2287.165} C_VEL
LIN {X 0,Y 573.246,Z 350.079,A -85,B 0,C 180,E1 -2289.606,E2 -2289.606} C_VEL
LIN {X 0,Y 573.236,Z 350.075,A -85,B 0,C 180,E1 -2292.641,E2 -2292.641} C_VEL
LIN {X 0,Y 573.234,Z 350.083,A -85,B 0,C 180,E1 -2295.666,E2 -2295.666} C_VEL
LIN {X 0,Y 573.239,Z 350.074,A -85,B 0,C 180,E1 -2298.544,E2 -2298.544} C_VEL
LIN {X 0,Y 573.243,Z 350.078,A -85,B 0,C 180,E1 -2301.298,E2 -2301.298} C_VEL
